C07312=1222.254,171.047,-53.911,-177.755,5.929,148.387
C07313=1222.250,171.296,-53.933,-177.752,5.931,148.387
C07314=1222.244,171.545,-53.955,-177.749,5.933,148.387
C07315=1222.240,171.794,-53.978,-177.747,5.934,148.386
C07316=1222.236,172.043,-54.000,-177.744,5.935,148.386
C07317=1222.230,172.292,-54.022,-177.742,5.936,148.385
C07318=1222.226,172.541,-54.044,-177.739,5.938,148.385
C07319=1222.221,172.789,-54.067,-177.736,5.940,148.384
C07320=1222.216,173.039,-54.089,-177.734,5.941,148.384
C07321=1222.212,173.288,-54.111,-177.732,5.943,148.384
C07322=1222.208,173.536,-54.134,-177.729,5.944,148.383
C07323=1222.203,173.786,-54.156,-177.726,5.945,148.383
C07324=1222.198,174.034,-54.179,-177.724,5.947,148.382
C07325=1222.194,174.283,-54.201,-177.721,5.949,148.382
C07326=1222.189,174.533,-54.223,-177.719,5.950,148.382
C07327=1222.184,174.781,-54.246,-177.716,5.951,148.381
C07328=1222.180,175.030,-54.268,-177.713,5.953,148.381
C07329=1222.174,175.279,-54.290,-177.711,5.954,148.380
C07330=1222.170,175.528,-54.313,-177.708,5.956,148.380
C07331=1222.165,175.778,-54.336,-177.706,5.957,148.379
C07332=1222.161,176.026,-54.358,-177.703,5.958,148.379
C07333=1222.157,176.275,-54.380,-177.701,5.960,148.379
C07334=1222.152,176.524,-54.403,-177.698,5.961,148.378
C07335=1222.147,176.773,-54.425,-177.696,5.963,148.378
C07336=1222.142,177.022,-54.448,-177.693,5.965,148.377
C07337=1222.138,177.271,-54.470,-177.691,5.966,148.377
C07338=1222.133,177.519,-54.493,-177.688,5.967,148.377
C07339=1222.128,177.769,-54.516,-177.685,5.969,148.376
C07340=1222.124,178.017,-54.538,-177.683,5.970,148.376
C07341=1222.119,178.266,-54.561,-177.680,5.972,148.375
C07342=1222.115,178.515,-54.583,-177.677,5.973,148.375
C07343=1222.110,178.765,-54.606,-177.675,5.974,148.375
C07344=1222.105,179.013,-54.628,-177.673,5.976,148.374
C07345=1222.101,179.262,-54.652,-177.669,5.978,148.374
C07346=1222.096,179.511,-54.674,-177.667,5.979,148.373
C07347=1222.092,179.760,-54.697,-177.665,5.981,148.373
C07348=1222.087,180.009,-54.719,-177.662,5.982,148.372
C07349=1222.082,180.258,-54.742,-177.659,5.984,148.372
C07350=1222.078,180.507,-54.765,-177.657,5.985,148.372
C07351=1222.073,180.756,-54.788,-177.654,5.987,148.371
C07352=1222.068,181.005,-54.811,-177.652,5.989,148.371
C07353=1222.064,181.254,-54.833,-177.649,5.990,148.370
C07354=1222.059,181.503,-54.856,-177.647,5.991,148.370
C07355=1222.054,181.751,-54.878,-177.644,5.993,148.370
C07356=1222.050,182.000,-54.902,-177.642,5.994,148.369
C07357=1222.045,182.249,-54.924,-177.639,5.996,148.369
C07358=1222.041,182.498,-54.947,-177.636,5.998,148.368
C07359=1222.037,182.747,-54.970,-177.634,5.999,148.368
C07360=1222.031,182.996,-54.992,-177.631,6.000,148.367
C07361=1222.026,183.245,-55.016,-177.628,6.002,148.367
C07362=1222.022,183.494,-55.038,-177.626,6.004,148.367
C07363=1222.018,183.743,-55.062,-177.624,6.005,148.366
C07364=1222.012,183.992,-55.084,-177.621,6.007,148.366
C07365=1222.008,184.240,-55.107,-177.618,6.009,148.366
C07366=1222.003,184.489,-55.130,-177.616,6.009,148.365
C07367=1221.999,184.738,-55.153,-177.613,6.011,148.365
C07368=1221.995,184.987,-55.176,-177.610,6.013,148.364
C07369=1221.989,185.257,-55.201,-177.608,6.015,148.364
C07370=1221.985,185.526,-55.226,-177.605,6.016,148.363
C07371=1221.980,185.796,-55.251,-177.602,6.018,148.363
C07372=1221.974,186.066,-55.276,-177.599,6.020,148.363
C07373=1221.970,186.315,-55.299,-177.597,6.021,148.362
C07374=1221.965,186.563,-55.322,-177.594,6.022,148.362
C07375=1221.960,186.812,-55.345,-177.592,6.024,148.361
C07376=1221.956,187.061,-55.368,-177.589,6.026,148.361
C07377=1221.951,187.310,-55.390,-177.587,6.027,148.361
C07378=1221.947,187.559,-55.414,-177.584,6.029,148.360
C07379=1221.942,187.809,-55.437,-177.581,6.031,148.360
C07380=1221.938,188.057,-55.460,-177.579,6.031,148.359
C07381=1221.933,188.306,-55.483,-177.576,6.033,148.359
C07382=1221.928,188.555,-55.506,-177.574,6.035,148.359
C07383=1221.923,188.804,-55.529,-177.571,6.037,148.358
C07384=1221.919,189.052,-55.552,-177.569,6.038,148.358
C07385=1221.915,189.301,-55.576,-177.566,6.040,148.358
C07386=1221.910,189.550,-55.599,-177.564,6.042,148.357
C07387=1221.905,189.799,-55.622,-177.560,6.043,148.357
C07388=1221.900,190.048,-55.646,-177.558,6.044,148.356
C07389=1221.896,190.296,-55.668,-177.556,6.046,148.356
C07390=1221.891,190.546,-55.691,-177.553,6.048,148.356
C07391=1221.887,190.795,-55.715,-177.550,6.050,148.355
C07392=1221.882,191.044,-55.738,-177.548,6.051,148.355
C07393=1221.877,191.293,-55.761,-177.546,6.052,148.355
C07394=1221.872,191.542,-55.785,-177.543,6.054,148.354
C07395=1221.869,191.790,-55.808,-177.540,6.056,148.354
C07396=1221.864,192.039,-55.832,-177.538,6.057,148.353
C07397=1221.859,192.288,-55.855,-177.535,6.059,148.353
C07398=1221.855,192.537,-55.878,-177.533,6.060,148.353
C07399=1221.850,192.786,-55.902,-177.530,6.062,148.352
C07400=1221.845,193.034,-55.925,-177.527,6.064,148.352
C07401=1221.840,193.283,-55.948,-177.525,6.065,148.351
C07402=1221.836,193.532,-55.972,-177.522,6.067,148.351
C07403=1221.831,193.781,-55.996,-177.519,6.069,148.351
C07404=1221.827,194.029,-56.018,-177.517,6.070,148.350
C07405=1221.822,194.278,-56.042,-177.515,6.071,148.350
C07406=1221.818,194.527,-56.065,-177.512,6.073,148.350
C07407=1221.813,194.776,-56.089,-177.509,6.075,148.349
C07408=1221.808,195.025,-56.112,-177.507,6.077,148.349
C07409=1221.804,195.274,-56.136,-177.504,6.079,148.348
C07410=1221.799,195.523,-56.159,-177.502,6.080,148.348
C07411=1221.795,195.771,-56.183,-177.499,6.081,148.348
C07412=1221.790,196.020,-56.207,-177.496,6.083,148.347
C07413=1221.785,196.269,-56.230,-177.494,6.085,148.347
C07414=1221.781,196.519,-56.253,-177.492,6.086,148.346
C07415=1221.776,196.767,-56.277,-177.489,6.088,148.346
C07416=1221.771,197.016,-56.301,-177.486,6.090,148.346
C07417=1221.767,197.265,-56.324,-177.484,6.091,148.345
C07418=1221.762,197.513,-56.348,-177.481,6.093,148.345
C07419=1221.758,197.762,-56.372,-177.479,6.094,148.345
C07420=1221.753,198.011,-56.395,-177.476,6.096,148.344
C07421=1221.749,198.260,-56.419,-177.474,6.098,148.344
C07422=1221.744,198.509,-56.442,-177.470,6.100,148.343
C07423=1221.739,198.757,-56.466,-177.468,6.101,148.343
C07424=1221.735,199.006,-56.490,-177.466,6.102,148.343
C07425=1221.730,199.255,-56.513,-177.463,6.104,148.342
C07426=1221.726,199.504,-56.538,-177.460,6.106,148.342
C07427=1221.722,199.754,-56.561,-177.458,6.108,148.342
C07428=1221.717,200.002,-56.585,-177.455,6.110,148.341
C07429=1221.712,200.251,-56.608,-177.453,6.112,148.341
C07430=1221.707,200.500,-56.633,-177.450,6.113,148.341
C07431=1221.703,200.749,-56.656,-177.448,6.114,148.340
C07432=1221.698,200.997,-56.680,-177.445,6.116,148.340
C07433=1221.694,201.246,-56.704,-177.443,6.118,148.340
C07434=1221.689,201.495,-56.728,-177.440,6.120,148.339
C07435=1221.684,201.744,-56.751,-177.437,6.121,148.339
C07436=1221.680,201.992,-56.775,-177.435,6.123,148.338
C07437=1221.675,202.241,-56.799,-177.432,6.124,148.338
C07438=1221.671,202.490,-56.824,-177.429,6.126,148.338
C07439=1221.666,202.740,-56.847,-177.427,6.128,148.337
C07440=1221.662,202.988,-56.871,-177.424,6.130,148.337
C07441=1221.657,203.237,-56.895,-177.422,6.131,148.337
C07442=1221.653,203.485,-56.919,-177.419,6.133,148.336
C07443=1221.648,203.734,-56.943,-177.417,6.135,148.336
C07444=1221.643,203.983,-56.967,-177.414,6.136,148.336
C07445=1221.639,204.232,-56.991,-177.411,6.138,148.335
C07446=1221.635,204.481,-57.015,-177.409,6.140,148.335
C07447=1221.630,204.730,-57.039,-177.407,6.141,148.335
C07448=1221.626,204.978,-57.063,-177.404,6.143,148.334
C07449=1221.620,205.227,-57.087,-177.401,6.145,148.334
C07450=1221.616,205.476,-57.111,-177.399,6.147,148.334
C07451=1221.611,205.724,-57.135,-177.396,6.149,148.333
C07452=1221.608,205.973,-57.159,-177.394,6.150,148.333
C07453=1221.602,206.223,-57.183,-177.391,6.152,148.333
C07454=1221.598,206.471,-57.207,-177.388,6.153,148.332
C07455=1221.593,206.720,-57.231,-177.386,6.155,148.332
C07456=1221.589,206.969,-57.255,-177.383,6.157,148.331
C07457=1221.584,207.218,-57.280,-177.380,6.158,148.331
C07458=1221.580,207.466,-57.304,-177.378,6.160,148.331
C07459=1221.575,207.715,-57.328,-177.375,6.162,148.330
C07460=1221.570,207.964,-57.352,-177.373,6.164,148.330
C07461=1221.565,208.213,-57.376,-177.370,6.165,148.330
C07462=1221.562,208.462,-57.400,-177.368,6.167,148.329
C07463=1221.557,208.710,-57.425,-177.365,6.169,148.329
C07464=1221.552,208.959,-57.449,-177.363,6.171,148.329
C07465=1221.548,209.207,-57.473,-177.360,6.172,148.328
C07466=1221.542,209.457,-57.497,-177.357,6.174,148.328
C07467=1221.538,209.706,-57.521,-177.355,6.176,148.328
C07468=1221.534,209.954,-57.546,-177.352,6.178,148.327
C07469=1221.529,210.203,-57.570,-177.349,6.180,148.327
C07470=1221.525,210.451,-57.594,-177.347,6.181,148.326
C07471=1221.520,210.701,-57.619,-177.345,6.183,148.326
C07472=1221.516,210.949,-57.643,-177.342,6.185,148.326
C07473=1221.510,211.219,-57.670,-177.339,6.186,148.325
C07474=1221.505,211.490,-57.696,-177.337,6.188,148.325
C07475=1221.501,211.761,-57.723,-177.334,6.191,148.325
C07476=1221.496,212.031,-57.749,-177.330,6.192,148.324
C07477=1221.491,212.280,-57.774,-177.328,6.194,148.324
C07478=1221.487,212.528,-57.798,-177.325,6.196,148.324
C07479=1221.482,212.777,-57.823,-177.323,6.197,148.323
C07480=1221.478,213.026,-57.847,-177.320,6.199,148.323
C07481=1221.473,213.274,-57.871,-177.318,6.201,148.323
C07482=1221.469,213.524,-57.896,-177.315,6.203,148.322
C07483=1221.464,213.772,-57.920,-177.313,6.205,148.322
C07484=1221.459,214.021,-57.945,-177.310,6.206,148.322
C07485=1221.455,214.270,-57.969,-177.307,6.208,148.321
C07486=1221.450,214.519,-57.994,-177.305,6.210,148.321
C07487=1221.446,214.767,-58.018,-177.302,6.212,148.321
C07488=1221.441,215.016,-58.043,-177.299,6.214,148.320
C07489=1221.437,215.265,-58.067,-177.297,6.216,148.320
C07490=1221.432,215.514,-58.092,-177.295,6.217,148.320
C07491=1221.428,215.762,-58.117,-177.293,6.219,148.319
C07492=1221.423,216.011,-58.142,-177.290,6.221,148.319
C07493=1221.418,216.259,-58.166,-177.287,6.223,148.319
C07494=1221.414,216.509,-58.191,-177.285,6.225,148.318
C07495=1221.409,216.757,-58.216,-177.282,6.226,148.318
C07496=1221.405,217.006,-58.240,-177.279,6.228,148.318
C07497=1221.400,217.255,-58.265,-177.277,6.230,148.317
C07498=1221.396,217.503,-58.289,-177.274,6.232,148.317
C07499=1221.391,217.752,-58.314,-177.271,6.234,148.317
C07500=1221.386,218.001,-58.339,-177.269,6.236,148.316
C07501=1221.382,218.250,-58.363,-177.266,6.237,148.316
C07502=1221.378,218.498,-58.389,-177.264,6.239,148.316
C07503=1221.373,218.747,-58.413,-177.262,6.240,148.315
C07504=1221.368,218.995,-58.438,-177.259,6.242,148.315
C07505=1221.364,219.245,-58.463,-177.256,6.244,148.315
C07506=1221.360,219.493,-58.488,-177.254,6.246,148.314
C07507=1221.355,219.742,-58.513,-177.251,6.248,148.314
C07508=1221.350,219.991,-58.537,-177.248,6.250,148.314
C07509=1221.347,220.239,-58.562,-177.246,6.252,148.313
C07510=1221.341,220.488,-58.587,-177.243,6.253,148.313
C07511=1221.336,220.737,-58.612,-177.240,6.255,148.313
C07512=1221.333,220.985,-58.637,-177.238,6.257,148.313
C07513=1221.328,221.234,-58.662,-177.236,6.259,148.312
C07514=1221.323,221.483,-58.687,-177.233,6.261,148.312
C07515=1221.319,221.731,-58.711,-177.230,6.263,148.312
C07516=1221.314,221.981,-58.736,-177.228,6.265,148.311
C07517=1221.310,222.229,-58.762,-177.225,6.267,148.311
C07518=1221.305,222.478,-58.787,-177.223,6.269,148.311
C07519=1221.301,222.727,-58.811,-177.220,6.270,148.310
C07520=1221.297,222.975,-58.837,-177.218,6.271,148.310
C07521=1221.291,223.224,-58.861,-177.215,6.273,148.310
C07522=1221.287,223.473,-58.887,-177.213,6.275,148.309
C07523=1221.283,223.721,-58.911,-177.210,6.277,148.309
C07524=1221.279,223.970,-58.937,-177.207,6.279,148.309
C07525=1221.273,224.219,-58.962,-177.205,6.281,148.309
C07526=1221.269,224.468,-58.987,-177.203,6.283,148.308
C07527=1221.265,224.716,-59.011,-177.200,6.285,148.308
C07528=1221.261,224.965,-59.037,-177.197,6.287,148.308
C07529=1221.255,225.214,-59.062,-177.195,6.288,148.307
C07530=1221.251,225.462,-59.088,-177.192,6.290,148.307
C07531=1221.246,225.711,-59.112,-177.189,6.292,148.307
C07532=1221.242,225.960,-59.138,-177.187,6.294,148.306
C07533=1221.238,226.208,-59.163,-177.184,6.296,148.306
C07534=1221.233,226.457,-59.188,-177.182,6.298,148.306
C07535=1221.228,226.705,-59.213,-177.179,6.300,148.306
C07536=1221.224,226.955,-59.238,-177.177,6.302,148.305
C07537=1221.219,227.203,-59.264,-177.174,6.304,148.305
C07538=1221.215,227.452,-59.289,-177.172,6.306,148.305
C07539=1221.210,227.701,-59.314,-177.169,6.307,148.304
C07540=1221.206,227.949,-59.339,-177.166,6.309,148.304
C07541=1221.202,228.198,-59.365,-177.164,6.311,148.304
C07542=1221.197,228.446,-59.390,-177.161,6.313,148.303
C07543=1221.193,228.695,-59.415,-177.159,6.315,148.303
C07544=1221.188,228.943,-59.441,-177.156,6.317,148.303
C07545=1221.183,229.193,-59.466,-177.154,6.319,148.303
C07546=1221.179,229.441,-59.492,-177.151,6.321,148.302
C07547=1221.174,229.690,-59.517,-177.149,6.322,148.302
C07548=1221.170,229.938,-59.543,-177.146,6.324,148.302
C07549=1221.165,230.187,-59.567,-177.144,6.326,148.301
C07550=1221.161,230.436,-59.593,-177.141,6.327,148.301
C07551=1221.156,230.685,-59.619,-177.139,6.330,148.301
C07552=1221.152,230.933,-59.644,-177.136,6.331,148.301
C07553=1221.147,231.182,-59.669,-177.134,6.333,148.300
C07554=1221.142,231.430,-59.695,-177.131,6.335,148.300
C07555=1221.138,231.679,-59.720,-177.128,6.337,148.300
C07556=1221.134,231.928,-59.746,-177.126,6.339,148.299
C07557=1221.129,232.176,-59.772,-177.124,6.341,148.299
C07558=1221.125,232.425,-59.797,-177.121,6.343,148.299
C07559=1221.120,232.674,-59.822,-177.118,6.345,148.299
C07560=1221.115,232.922,-59.848,-177.116,6.347,148.298
C07561=1221.111,233.171,-59.873,-177.113,6.349,148.298
C07562=1221.107,233.420,-59.899,-177.111,6.350,148.298
C07563=1221.102,233.668,-59.925,-177.108,6.353,148.297
C07564=1221.098,233.917,-59.950,-177.106,6.354,148.297
C07565=1221.094,234.166,-59.976,-177.103,6.356,148.297
C07566=1221.089,234.414,-60.002,-177.101,6.358,148.297
C07567=1221.085,234.663,-60.027,-177.098,6.360,148.296
C07568=1221.080,234.911,-60.053,-177.095,6.362,148.296
C07569=1221.076,235.159,-60.078,-177.093,6.364,148.296
C07570=1221.071,235.409,-60.105,-177.090,6.366,148.295
C07571=1221.066,235.657,-60.130,-177.088,6.368,148.295
C07572=1221.062,235.906,-60.156,-177.085,6.370,148.295
C07573=1221.057,236.154,-60.182,-177.083,6.372,148.295
C07574=1221.053,236.403,-60.207,-177.080,6.374,148.294
C07575=1221.049,236.652,-60.233,-177.078,6.376,148.294
C07576=1221.044,236.900,-60.259,-177.075,6.377,148.294
C07577=1221.039,237.172,-60.287,-177.072,6.380,148.293
C07578=1221.035,237.443,-60.315,-177.069,6.382,148.293
C07579=1221.029,237.715,-60.344,-177.067,6.384,148.293
C07580=1221.024,237.987,-60.372,-177.064,6.387,148.293
C07581=1221.020,238.235,-60.397,-177.061,6.388,148.292
C07582=1221.015,238.484,-60.423,-177.058,6.390,148.292
C07583=1221.011,238.732,-60.449,-177.056,6.393,148.292
C07584=1221.007,238.981,-60.475,-177.054,6.394,148.292
C07585=1221.002,239.230,-60.501,-177.051,6.396,148.291
C07586=1220.997,239.478,-60.527,-177.048,6.398,148.291
C07587=1220.993,239.727,-60.552,-177.046,6.400,148.291
C07588=1220.989,239.975,-60.578,-177.044,6.402,148.290
C07589=1220.984,240.224,-60.605,-177.041,6.404,148.290
C07590=1220.979,240.472,-60.631,-177.038,6.406,148.290
C07591=1220.975,240.721,-60.656,-177.036,6.408,148.290
C07592=1220.971,240.970,-60.682,-177.034,6.410,148.289
C07593=1220.966,241.218,-60.709,-177.031,6.412,148.289
C07594=1220.962,241.467,-60.735,-177.028,6.414,148.289
C07595=1220.957,241.715,-60.760,-177.026,6.416,148.289
C07596=1220.952,241.964,-60.787,-177.024,6.418,148.288
C07597=1220.948,242.212,-60.813,-177.021,6.420,148.288
C07598=1220.944,242.461,-60.839,-177.018,6.422,148.288
C07599=1220.939,242.710,-60.865,-177.016,6.423,148.287
C07600=1220.935,242.958,-60.892,-177.014,6.426,148.287
C07601=1220.930,243.206,-60.917,-177.011,6.427,148.287
C07602=1220.925,243.456,-60.943,-177.008,6.429,148.287
C07603=1220.921,243.704,-60.970,-177.005,6.432,148.286
C07604=1220.917,243.953,-60.996,-177.003,6.434,148.286
C07605=1220.912,244.202,-61.022,-177.001,6.436,148.286
C07606=1220.908,244.450,-61.048,-176.998,6.438,148.286
C07607=1220.904,244.699,-61.074,-176.995,6.440,148.285
C07608=1220.899,244.946,-61.101,-176.993,6.442,148.285
C07609=1220.895,245.195,-61.127,-176.991,6.444,148.285
C07610=1220.890,245.444,-61.153,-176.988,6.446,148.285
C07611=1220.886,245.693,-61.179,-176.985,6.448,148.284
C07612=1220.882,245.941,-61.205,-176.983,6.450,148.284
C07613=1220.877,246.190,-61.232,-176.981,6.452,148.284
C07614=1220.873,246.439,-61.258,-176.978,6.454,148.284
C07615=1220.868,246.687,-61.285,-176.975,6.455,148.283
C07616=1220.864,246.936,-61.311,-176.973,6.458,148.283
C07617=1220.859,247.184,-61.338,-176.971,6.459,148.283
C07618=1220.854,247.433,-61.363,-176.967,6.462,148.283
C07619=1220.850,247.681,-61.390,-176.965,6.464,148.283
C07620=1220.845,247.930,-61.416,-176.963,6.466,148.282
C07621=1220.841,248.178,-61.443,-176.960,6.468,148.282
C07622=1220.837,248.427,-61.470,-176.957,6.470,148.282
C07623=1220.832,248.676,-61.496,-176.955,6.472,148.282
C07624=1220.828,248.924,-61.522,-176.953,6.474,148.281
C07625=1220.823,249.173,-61.549,-176.950,6.476,148.281
C07626=1220.819,249.421,-61.575,-176.948,6.478,148.281
C07627=1220.814,249.670,-61.602,-176.945,6.480,148.281
C07628=1220.810,249.918,-61.628,-176.943,6.482,148.280
C07629=1220.806,250.167,-61.655,-176.941,6.484,148.280
C07630=1220.801,250.416,-61.681,-176.937,6.487,148.280
C07631=1220.797,250.664,-61.708,-176.935,6.489,148.280
C07632=1220.793,250.912,-61.734,-176.932,6.491,148.279
C07633=1220.788,251.162,-61.761,-176.930,6.493,148.279
C07634=1220.783,251.410,-61.788,-176.927,6.495,148.279
C07635=1220.779,251.658,-61.814,-176.925,6.496,148.279
C07636=1220.775,251.907,-61.841,-176.923,6.499,148.279
C07637=1220.770,252.156,-61.867,-176.920,6.501,148.278
C07638=1220.766,252.404,-61.894,-176.917,6.502,148.278
C07639=1220.761,252.653,-61.921,-176.915,6.505,148.278
C07640=1220.757,252.901,-61.948,-176.912,6.507,148.278
C07641=1220.752,253.150,-61.974,-176.909,6.509,148.277
C07642=1220.748,253.398,-62.001,-176.907,6.511,148.277
C07643=1220.744,253.647,-62.028,-176.905,6.513,148.277
C07644=1220.739,253.895,-62.055,-176.902,6.515,148.277
C07645=1220.735,254.143,-62.081,-176.900,6.517,148.276
C07646=1220.730,254.392,-62.107,-176.897,6.519,148.276
C07647=1220.725,254.641,-62.135,-176.895,6.521,148.276
C07648=1220.721,254.889,-62.161,-176.892,6.524,148.276
C07649=1220.717,255.137,-62.188,-176.889,6.526,148.276
C07650=1220.712,255.386,-62.215,-176.887,6.528,148.275
C07651=1220.707,255.634,-62.242,-176.885,6.530,148.275
C07652=1220.704,255.883,-62.269,-176.882,6.532,148.275
C07653=1220.699,256.131,-62.296,-176.880,6.534,148.275
C07654=1220.694,256.380,-62.323,-176.877,6.536,148.274
C07655=1220.691,256.629,-62.350,-176.874,6.539,148.274
C07656=1220.686,256.878,-62.376,-176.872,6.541,148.274
C07657=1220.681,257.126,-62.403,-176.869,6.543,148.274
C07658=1220.677,257.375,-62.430,-176.867,6.545,148.273
C07659=1220.673,257.623,-62.457,-176.865,6.547,148.273
C07660=1220.668,257.871,-62.484,-176.862,6.549,148.273
C07661=1220.663,258.120,-62.511,-176.860,6.551,148.273
C07662=1220.659,258.368,-62.538,-176.857,6.553,148.273
C07663=1220.654,258.617,-62.565,-176.854,6.556,148.272
C07664=1220.651,258.866,-62.592,-176.852,6.558,148.272
C07665=1220.646,259.114,-62.619,-176.849,6.560,148.272
C07666=1220.642,259.362,-62.646,-176.847,6.561,148.272
C07667=1220.637,259.611,-62.674,-176.845,6.564,148.272
C07668=1220.632,259.859,-62.701,-176.842,6.566,148.271
C07669=1220.628,260.108,-62.728,-176.839,6.569,148.271
C07670=1220.624,260.356,-62.754,-176.837,6.570,148.271
C07671=1220.620,260.605,-62.782,-176.834,6.572,148.271
C07672=1220.615,260.853,-62.809,-176.832,6.575,148.271
C07673=1220.611,261.102,-62.836,-176.829,6.576,148.270
C07674=1220.606,261.350,-62.863,-176.827,6.579,148.270
C07675=1220.602,261.598,-62.890,-176.824,6.581,148.270
C07676=1220.597,261.847,-62.918,-176.822,6.583,148.270
C07677=1220.593,262.096,-62.945,-176.819,6.585,148.270
C07678=1220.589,262.344,-62.971,-176.817,6.587,148.269
C07679=1220.584,262.593,-62.999,-176.815,6.589,148.269
C07680=1220.580,262.841,-63.026,-176.812,6.591,148.269
C07681=1220.574,263.114,-63.056,-176.809,6.594,148.269
C07682=1220.570,263.386,-63.086,-176.807,6.596,148.269
C07683=1220.565,263.659,-63.116,-176.804,6.599,148.268
C07684=1220.561,263.932,-63.146,-176.801,6.601,148.268
C07685=1220.556,264.180,-63.173,-176.798,6.604,148.268
C07686=1220.552,264.428,-63.201,-176.796,6.606,148.268
C07687=1220.547,264.677,-63.228,-176.793,6.608,148.267
C07688=1220.543,264.926,-63.255,-176.791,6.610,148.267
C07689=1220.539,265.174,-63.283,-176.788,6.612,148.267
C07690=1220.534,265.422,-63.310,-176.786,6.614,148.267
C07691=1220.529,265.671,-63.337,-176.783,6.617,148.267
C07692=1220.525,265.919,-63.365,-176.781,6.619,148.267
C07693=1220.521,266.168,-63.392,-176.778,6.621,148.266
C07694=1220.516,266.416,-63.419,-176.776,6.623,148.266
C07695=1220.512,266.664,-63.447,-176.774,6.625,148.266
C07696=1220.508,266.913,-63.475,-176.771,6.628,148.266
C07697=1220.503,267.161,-63.502,-176.768,6.630,148.266
C07698=1220.499,267.410,-63.530,-176.766,6.632,148.265
C07699=1220.493,267.658,-63.557,-176.764,6.634,148.265
C07700=1220.490,267.907,-63.585,-176.761,6.636,148.265
C07701=1220.485,268.156,-63.612,-176.758,6.639,148.265
C07702=1220.481,268.403,-63.640,-176.756,6.641,148.265
C07703=1220.477,268.653,-63.668,-176.754,6.643,148.265
C07704=1220.472,268.901,-63.695,-176.751,6.645,148.264
C07705=1220.468,269.149,-63.722,-176.748,6.648,148.264
C07706=1220.464,269.398,-63.751,-176.746,6.650,148.264
C07707=1220.459,269.646,-63.778,-176.744,6.652,148.264
C07708=1220.454,269.894,-63.806,-176.741,6.654,148.264
C07709=1220.450,270.143,-63.834,-176.739,6.656,148.263
C07710=1220.446,270.391,-63.861,-176.736,6.659,148.263
C07711=1220.441,270.639,-63.889,-176.734,6.661,148.263
C07712=1220.437,270.888,-63.916,-176.731,6.663,148.263
C07713=1220.433,271.136,-63.944,-176.729,6.665,148.263
C07714=1220.428,271.385,-63.971,-176.726,6.668,148.262
C07715=1220.424,271.634,-64.000,-176.724,6.670,148.262
C07716=1220.419,271.882,-64.028,-176.721,6.672,148.262
C07717=1220.415,272.130,-64.055,-176.719,6.674,148.262
C07718=1220.411,272.379,-64.083,-176.716,6.676,148.262
C07719=1220.406,272.627,-64.111,-176.714,6.679,148.262
C07720=1220.401,272.875,-64.138,-176.711,6.681,148.261
C07721=1220.397,273.124,-64.167,-176.709,6.683,148.261
C07722=1220.393,273.372,-64.194,-176.706,6.685,148.261
C07723=1220.389,273.620,-64.222,-176.704,6.688,148.261
C07724=1220.384,273.869,-64.250,-176.701,6.690,148.261
C07725=1220.380,274.117,-64.278,-176.699,6.692,148.261
C07726=1220.376,274.366,-64.306,-176.697,6.694,148.261
C07727=1220.371,274.614,-64.334,-176.694,6.697,148.260
C07728=1220.367,274.863,-64.362,-176.691,6.699,148.260
C07729=1220.362,275.111,-64.390,-176.689,6.701,148.260
C07730=1220.359,275.359,-64.418,-176.687,6.703,148.260
C07731=1220.354,275.608,-64.446,-176.684,6.706,148.260
C07732=1220.349,275.855,-64.474,-176.681,6.708,148.260
C07733=1220.345,276.105,-64.501,-176.679,6.710,148.259
C07734=1220.340,276.353,-64.530,-176.677,6.712,148.259
C07735=1220.336,276.601,-64.558,-176.674,6.715,148.259
C07736=1220.332,276.849,-64.586,-176.671,6.717,148.259
C07737=1220.327,277.098,-64.614,-176.669,6.719,148.259
C07738=1220.323,277.346,-64.642,-176.666,6.722,148.259
C07739=1220.319,277.595,-64.670,-176.664,6.724,148.258
C07740=1220.314,277.843,-64.699,-176.661,6.726,148.258
C07741=1220.310,278.092,-64.726,-176.659,6.728,148.258
C07742=1220.305,278.340,-64.754,-176.657,6.731,148.258
C07743=1220.301,278.589,-64.783,-176.654,6.733,148.258
C07744=1220.297,278.837,-64.810,-176.652,6.735,148.258
C07745=1220.293,279.086,-64.839,-176.649,6.737,148.257
C07746=1220.288,279.333,-64.867,-176.647,6.740,148.257
C07747=1220.284,279.582,-64.896,-176.644,6.743,148.257
C07748=1220.279,279.830,-64.923,-176.642,6.744,148.257
C07749=1220.275,280.079,-64.952,-176.639,6.748,148.257
C07750=1220.270,280.327,-64.980,-176.637,6.749,148.257
C07751=1220.267,280.576,-65.008,-176.634,6.752,148.257
C07752=1220.262,280.824,-65.036,-176.632,6.754,148.257
C07753=1220.258,281.072,-65.065,-176.629,6.757,148.256
C07754=1220.253,281.320,-65.094,-176.627,6.759,148.256
C07755=1220.249,281.568,-65.122,-176.625,6.761,148.256
C07756=1220.244,281.817,-65.150,-176.622,6.764,148.256
C07757=1220.241,282.065,-65.178,-176.620,6.766,148.256
C07758=1220.235,282.313,-65.207,-176.617,6.768,148.256
C07759=1220.232,282.562,-65.235,-176.615,6.770,148.256
C07760=1220.227,282.811,-65.264,-176.612,6.773,148.256
C07761=1220.223,283.059,-65.291,-176.610,6.775,148.255
C07762=1220.219,283.307,-65.321,-176.608,6.777,148.255
C07763=1220.214,283.555,-65.349,-176.605,6.780,148.255
C07764=1220.210,283.804,-65.377,-176.602,6.782,148.255
C07765=1220.205,284.052,-65.406,-176.600,6.784,148.255
C07766=1220.201,284.301,-65.434,-176.598,6.787,148.255
C07767=1220.197,284.549,-65.463,-176.595,6.789,148.254
C07768=1220.192,284.797,-65.491,-176.593,6.791,148.254
C07769=1220.188,285.046,-65.520,-176.591,6.794,148.254
C07770=1220.183,285.294,-65.548,-176.588,6.796,148.254
C07771=1220.179,285.542,-65.577,-176.585,6.799,148.254
C07772=1220.175,285.791,-65.606,-176.583,6.801,148.254
C07773=1220.170,286.039,-65.634,-176.580,6.803,148.254
C07774=1220.166,286.287,-65.663,-176.578,6.806,148.254
C07775=1220.162,286.536,-65.692,-176.576,6.808,148.254
C07776=1220.158,286.783,-65.720,-176.573,6.811,148.253
C07777=1220.153,287.032,-65.749,-176.571,6.813,148.253
C07778=1220.148,287.280,-65.777,-176.569,6.815,148.253
C07779=1220.145,287.529,-65.805,-176.566,6.818,148.253
C07780=1220.140,287.777,-65.835,-176.563,6.820,148.253
C07781=1220.135,288.025,-65.863,-176.561,6.822,148.253
C07782=1220.131,288.274,-65.892,-176.558,6.825,148.253
C07783=1220.127,288.522,-65.921,-176.556,6.827,148.253
C07784=1220.122,288.770,-65.949,-176.554,6.829,148.253
C07785=1220.117,289.044,-65.981,-176.551,6.832,148.252
C07786=1220.113,289.318,-66.013,-176.548,6.835,148.252
C07787=1220.108,289.592,-66.045,-176.546,6.837,148.252
C07788=1220.103,289.867,-66.077,-176.543,6.840,148.252
C07789=1220.099,290.115,-66.106,-176.541,6.842,148.252
C07790=1220.094,290.363,-66.134,-176.538,6.845,148.252
C07791=1220.091,290.611,-66.163,-176.536,6.847,148.252
C07792=1220.086,290.860,-66.192,-176.533,6.849,148.252
C07793=1220.082,291.108,-66.221,-176.530,6.852,148.252
C07794=1220.077,291.357,-66.250,-176.528,6.855,148.251
C07795=1220.073,291.605,-66.279,-176.526,6.857,148.251
C07796=1220.069,291.853,-66.307,-176.524,6.860,148.251
C07797=1220.064,292.101,-66.336,-176.521,6.862,148.251
C07798=1220.060,292.349,-66.366,-176.519,6.864,148.251
C07799=1220.056,292.598,-66.395,-176.516,6.867,148.251
C07800=1220.051,292.846,-66.424,-176.514,6.869,148.251
C07801=1220.047,293.094,-66.452,-176.511,6.872,148.251
C07802=1220.043,293.343,-66.481,-176.509,6.874,148.251
C07803=1220.039,293.591,-66.511,-176.507,6.876,148.251
C07804=1220.034,293.840,-66.540,-176.504,6.879,148.251
C07805=1220.030,294.088,-66.569,-176.502,6.882,148.251
C07806=1220.025,294.336,-66.598,-176.499,6.883,148.250
C07807=1220.021,294.584,-66.628,-176.497,6.887,148.250
C07808=1220.017,294.832,-66.656,-176.495,6.889,148.250
C07809=1220.013,295.081,-66.685,-176.492,6.891,148.250
C07810=1220.008,295.328,-66.714,-176.490,6.894,148.250
C07811=1220.004,295.577,-66.743,-176.487,6.896,148.250
C07812=1220.000,295.825,-66.772,-176.485,6.898,148.250
C07813=1219.995,296.074,-66.802,-176.482,6.901,148.250
C07814=1219.991,296.322,-66.831,-176.480,6.903,148.250
C07815=1219.987,296.570,-66.861,-176.478,6.906,148.250
C07816=1219.982,296.818,-66.889,-176.475,6.909,148.250
C07817=1219.978,297.067,-66.919,-176.473,6.910,148.249
C07818=1219.974,297.315,-66.948,-176.470,6.914,148.249
C07819=1219.969,297.563,-66.978,-176.468,6.916,148.249
C07820=1219.965,297.811,-67.007,-176.466,6.918,148.249
C07821=1219.961,298.060,-67.036,-176.463,6.921,148.249
C07822=1219.956,298.308,-67.065,-176.461,6.923,148.249
C07823=1219.952,298.556,-67.094,-176.459,6.926,148.249
C07824=1219.948,298.804,-67.124,-176.456,6.928,148.249
C07825=1219.943,299.053,-67.153,-176.454,6.930,148.249
C07826=1219.939,299.301,-67.183,-176.451,6.933,148.249
C07827=1219.935,299.549,-67.212,-176.449,6.936,148.249
C07828=1219.931,299.797,-67.242,-176.447,6.938,148.249
C07829=1219.926,300.045,-67.271,-176.444,6.941,148.249
C07830=1219.922,300.293,-67.300,-176.442,6.943,148.249
C07831=1219.918,300.542,-67.330,-176.439,6.946,148.249
C07832=1219.914,300.790,-67.359,-176.437,6.948,148.248
C07833=1219.909,301.038,-67.388,-176.435,6.950,148.248
C07834=1219.905,301.286,-67.418,-176.432,6.953,148.248
C07835=1219.901,301.535,-67.447,-176.430,6.955,148.248
C07836=1219.896,301.783,-67.477,-176.427,6.959,148.248
C07837=1219.892,302.032,-67.507,-176.425,6.961,148.248
C07838=1219.888,302.280,-67.536,-176.423,6.963,148.248
C07839=1219.884,302.528,-67.566,-176.420,6.966,148.248
C07840=1219.879,302.776,-67.595,-176.418,6.968,148.248
C07841=1219.875,303.024,-67.624,-176.416,6.971,148.248
C07842=1219.870,303.272,-67.654,-176.414,6.973,148.248
C07843=1219.865,303.521,-67.684,-176.411,6.976,148.248
C07844=1219.862,303.768,-67.714,-176.409,6.979,148.248
C07845=1219.857,304.017,-67.743,-176.407,6.981,148.248
C07846=1219.853,304.265,-67.773,-176.404,6.984,148.248
C07847=1219.849,304.513,-67.802,-176.402,6.986,148.248
C07848=1219.844,304.762,-67.832,-176.399,6.988,148.247
C07849=1219.840,305.010,-67.862,-176.397,6.991,148.247
C07850=1219.836,305.258,-67.892,-176.394,6.993,148.247
C07851=1219.832,305.506,-67.921,-176.392,6.996,148.247
C07852=1219.828,305.754,-67.951,-176.390,6.999,148.247
C07853=1219.823,306.003,-67.981,-176.388,7.001,148.247
C07854=1219.819,306.250,-68.011,-176.385,7.004,148.247
C07855=1219.815,306.499,-68.041,-176.383,7.006,148.247
C07856=1219.811,306.747,-68.070,-176.380,7.009,148.247
C07857=1219.806,306.996,-68.100,-176.378,7.011,148.247
C07858=1219.802,307.243,-68.130,-176.376,7.014,148.247
C07859=1219.798,307.491,-68.160,-176.373,7.017,148.247
C07860=1219.793,307.740,-68.190,-176.371,7.019,148.247
C07861=1219.789,307.988,-68.220,-176.368,7.022,148.247
C07862=1219.785,308.236,-68.249,-176.367,7.024,148.247
C07863=1219.780,308.485,-68.279,-176.365,7.027,148.247
C07864=1219.776,308.732,-68.310,-176.362,7.030,148.247
C07865=1219.772,308.980,-68.339,-176.360,7.032,148.247
C07866=1219.767,309.229,-68.369,-176.357,7.035,148.247
C07867=1219.763,309.477,-68.399,-176.355,7.037,148.247
C07868=1219.759,309.725,-68.429,-176.352,7.040,148.247
C07869=1219.754,309.973,-68.459,-176.350,7.042,148.247
C07870=1219.750,310.221,-68.489,-176.348,7.045,148.247
C07871=1219.746,310.469,-68.519,-176.346,7.048,148.247
C07872=1219.741,310.717,-68.549,-176.343,7.050,148.247
C07873=1219.737,310.966,-68.579,-176.341,7.053,148.247
C07874=1219.733,311.214,-68.610,-176.339,7.055,148.247
C07875=1219.729,311.463,-68.639,-176.336,7.058,148.247
C07876=1219.725,311.710,-68.669,-176.334,7.060,148.247
C07877=1219.720,311.959,-68.699,-176.332,7.063,148.247
C07878=1219.716,312.206,-68.730,-176.330,7.066,148.247
C07879=1219.711,312.454,-68.760,-176.328,7.068,148.247
C07880=1219.707,312.703,-68.790,-176.325,7.071,148.247
C07881=1219.703,312.951,-68.821,-176.323,7.073,148.247
C07882=1219.698,313.199,-68.850,-176.321,7.076,148.247
C07883=1219.695,313.447,-68.881,-176.318,7.079,148.247
C07884=1219.690,313.696,-68.911,-176.316,7.081,148.247
C07885=1219.686,313.943,-68.941,-176.314,7.084,148.247
C07886=1219.682,314.191,-68.971,-176.312,7.086,148.247
C07887=1219.678,314.440,-69.001,-176.309,7.090,148.247
C07888=1219.673,314.688,-69.032,-176.307,7.092,148.247
C07889=1219.668,314.964,-69.065,-176.304,7.095,148.247
C07890=1219.664,315.240,-69.099,-176.301,7.098,148.247
C07891=1219.659,315.516,-69.133,-176.299,7.100,148.247
C07892=1219.654,315.792,-69.167,-176.297,7.103,148.247
C07893=1219.650,316.039,-69.197,-176.294,7.106,148.247
C07894=1219.645,316.288,-69.227,-176.292,7.109,148.247
C07895=1219.641,316.536,-69.257,-176.290,7.112,148.247
C07896=1219.637,316.784,-69.288,-176.288,7.114,148.247
C07897=1219.633,317.032,-69.318,-176.285,7.116,148.247
C07898=1219.628,317.280,-69.349,-176.283,7.119,148.247
C07899=1219.625,317.528,-69.379,-176.281,7.122,148.247
C07900=1219.620,317.776,-69.409,-176.279,7.125,148.247
C07901=1219.616,318.025,-69.441,-176.276,7.127,148.247
C07902=1219.612,318.272,-69.471,-176.274,7.130,148.247
C07903=1219.607,318.521,-69.501,-176.272,7.133,148.247
C07904=1219.603,318.769,-69.532,-176.269,7.136,148.247
C07905=1219.599,319.017,-69.562,-176.267,7.138,148.247
C07906=1219.595,319.265,-69.593,-176.265,7.140,148.247
C07907=1219.591,319.513,-69.623,-176.263,7.143,148.247
C07908=1219.586,319.761,-69.654,-176.261,7.146,148.247
C07909=1219.582,320.009,-69.685,-176.258,7.149,148.247
C07910=1219.578,320.257,-69.715,-176.256,7.151,148.247
C07911=1219.573,320.506,-69.745,-176.254,7.154,148.247
C07912=1219.569,320.754,-69.776,-176.252,7.156,148.247
C07913=1219.565,321.001,-69.806,-176.250,7.159,148.247
C07914=1219.561,321.250,-69.837,-176.247,7.162,148.247
C07915=1219.556,321.498,-69.868,-176.245,7.164,148.247
C07916=1219.552,321.746,-69.899,-176.243,7.167,148.247
C07917=1219.548,321.994,-69.929,-176.241,7.169,148.247
C07918=1219.544,322.242,-69.960,-176.238,7.173,148.248
C07919=1219.539,322.490,-69.991,-176.236,7.175,148.248
C07920=1219.535,322.738,-70.021,-176.234,7.178,148.248
C07921=1219.531,322.986,-70.052,-176.232,7.181,148.248
C07922=1219.527,323.234,-70.083,-176.230,7.183,148.248
C07923=1219.522,323.482,-70.114,-176.227,7.186,148.248
C07924=1219.519,323.730,-70.145,-176.226,7.188,148.248
C07925=1219.514,323.978,-70.176,-176.223,7.191,148.248
C07926=1219.510,324.226,-70.206,-176.221,7.194,148.248
C07927=1219.506,324.475,-70.238,-176.219,7.197,148.248
C07928=1219.501,324.723,-70.268,-176.217,7.199,148.248
C07929=1219.497,324.970,-70.298,-176.214,7.201,148.248
C07930=1219.493,325.219,-70.330,-176.212,7.205,148.248
C07931=1219.489,325.467,-70.360,-176.210,7.207,148.248
C07932=1219.484,325.715,-70.391,-176.208,7.210,148.248
C07933=1219.480,325.963,-70.423,-176.206,7.213,148.248
C07934=1219.476,326.211,-70.454,-176.203,7.216,148.248
C07935=1219.472,326.459,-70.484,-176.202,7.218,148.248
C07936=1219.468,326.707,-70.515,-176.199,7.221,148.248
C07937=1219.463,326.955,-70.546,-176.197,7.224,148.249
C07938=1219.459,327.202,-70.577,-176.195,7.226,148.249
C07939=1219.455,327.451,-70.608,-176.193,7.229,148.249
C07940=1219.450,327.699,-70.639,-176.191,7.232,148.249
C07941=1219.446,327.948,-70.670,-176.188,7.235,148.249
C07942=1219.442,328.195,-70.702,-176.187,7.237,148.249
C07943=1219.438,328.443,-70.732,-176.184,7.240,148.249
C07944=1219.434,328.691,-70.763,-176.182,7.243,148.249
C07945=1219.430,328.939,-70.795,-176.180,7.246,148.249
C07946=1219.426,329.187,-70.826,-176.178,7.248,148.249
C07947=1219.421,329.435,-70.856,-176.176,7.250,148.249
C07948=1219.417,329.683,-70.888,-176.174,7.254,148.249
C07949=1219.413,329.931,-70.919,-176.172,7.256,148.249
C07950=1219.408,330.179,-70.950,-176.169,7.259,148.250
C07951=1219.405,330.427,-70.982,-176.167,7.262,148.250
C07952=1219.400,330.675,-71.012,-176.165,7.265,148.250
C07953=1219.396,330.923,-71.044,-176.163,7.267,148.250
C07954=1219.392,331.171,-71.075,-176.161,7.270,148.250
C07955=1219.387,331.419,-71.106,-176.159,7.273,148.250
C07956=1219.383,331.667,-71.138,-176.157,7.275,148.250
C07957=1219.379,331.915,-71.168,-176.154,7.278,148.250
C07958=1219.375,332.163,-71.200,-176.153,7.281,148.250
C07959=1219.370,332.411,-71.231,-176.150,7.284,148.250
C07960=1219.367,332.659,-71.263,-176.148,7.286,148.251
C07961=1219.362,332.907,-71.294,-176.147,7.289,148.251
C07962=1219.358,333.155,-71.325,-176.144,7.292,148.251
C07963=1219.354,333.403,-71.356,-176.142,7.295,148.251
C07964=1219.350,333.651,-71.388,-176.140,7.298,148.251
C07965=1219.345,333.899,-71.419,-176.138,7.300,148.251
C07966=1219.341,334.148,-71.451,-176.136,7.303,148.251
C07967=1219.336,334.396,-71.482,-176.134,7.306,148.251
C07968=1219.333,334.644,-71.514,-176.132,7.309,148.251
C07969=1219.328,334.892,-71.545,-176.130,7.311,148.251
C07970=1219.324,335.140,-71.577,-176.128,7.314,148.252
C07971=1219.320,335.387,-71.608,-176.126,7.317,148.252
C07972=1219.316,335.636,-71.639,-176.124,7.319,148.252
C07973=1219.312,335.883,-71.671,-176.121,7.323,148.252
C07974=1219.308,336.131,-71.702,-176.119,7.325,148.252
C07975=1219.303,336.379,-71.734,-176.117,7.328,148.252
C07976=1219.299,336.627,-71.766,-176.116,7.331,148.252
C07977=1219.295,336.875,-71.797,-176.113,7.333,148.252
C07978=1219.291,337.123,-71.828,-176.111,7.336,148.253
C07979=1219.286,337.371,-71.860,-176.110,7.339,148.253
C07980=1219.283,337.619,-71.892,-176.107,7.342,148.253
C07981=1219.277,337.867,-71.923,-176.105,7.345,148.253
C07982=1219.274,338.115,-71.955,-176.104,7.347,148.253
C07983=1219.270,338.363,-71.987,-176.101,7.350,148.253
C07984=1219.266,338.610,-72.018,-176.099,7.353,148.253
C07985=1219.262,338.859,-72.049,-176.097,7.356,148.254
C07986=1219.257,339.107,-72.081,-176.096,7.358,148.254
C07987=1219.253,339.355,-72.113,-176.093,7.362,148.254
C07988=1219.249,339.603,-72.145,-176.091,7.364,148.254
C07989=1219.244,339.851,-72.176,-176.090,7.367,148.254
C07990=1219.240,340.099,-72.208,-176.087,7.370,148.254
C07991=1219.236,340.346,-72.240,-176.086,7.372,148.254
C07992=1219.232,340.594,-72.272,-176.083,7.376,148.254
C07993=1219.228,340.872,-72.307,-176.081,7.378,148.255
C07994=1219.222,341.150,-72.343,-176.079,7.381,148.255
C07995=1219.218,341.428,-72.378,-176.077,7.385,148.255
C07996=1219.213,341.706,-72.414,-176.074,7.388,148.255
C07997=1219.209,341.954,-72.446,-176.073,7.390,148.255
C07998=1219.205,342.202,-72.477,-176.071,7.394,148.256
C07999=1219.200,342.450,-72.509,-176.069,7.396,148.256
C08000=1219.196,342.697,-72.541,-176.067,7.400,148.256
C08001=1219.192,342.945,-72.573,-176.065,7.402,148.256
C08002=1219.188,343.194,-72.605,-176.063,7.404,148.256
C08003=1219.183,343.441,-72.637,-176.061,7.408,148.256
C08004=1219.180,343.689,-72.669,-176.059,7.410,148.257
C08005=1219.175,343.938,-72.701,-176.057,7.414,148.257
C08006=1219.171,344.185,-72.732,-176.055,7.416,148.257
C08007=1219.167,344.433,-72.765,-176.054,7.419,148.257
C08008=1219.163,344.681,-72.797,-176.052,7.422,148.257
C08009=1219.159,344.929,-72.828,-176.049,7.424,148.257
C08010=1219.154,345.177,-72.861,-176.047,7.428,148.258
C08011=1219.150,345.425,-72.893,-176.046,7.430,148.258
C08012=1219.145,345.673,-72.925,-176.044,7.433,148.258
C08013=1219.142,345.921,-72.956,-176.042,7.436,148.258
C08014=1219.138,346.168,-72.989,-176.040,7.438,148.258
C08015=1219.133,346.416,-73.021,-176.038,7.442,148.259
C08016=1219.129,346.664,-73.053,-176.036,7.444,148.259
C08017=1219.125,346.912,-73.085,-176.035,7.447,148.259
C08018=1219.121,347.160,-73.117,-176.032,7.450,148.259
C08019=1219.116,347.408,-73.149,-176.031,7.453,148.259
C08020=1219.113,347.656,-73.181,-176.029,7.455,148.259
C08021=1219.108,347.904,-73.214,-176.027,7.459,148.260
C08022=1219.104,348.151,-73.246,-176.025,7.461,148.260
C08023=1219.100,348.399,-73.278,-176.023,7.464,148.260
C08024=1219.096,348.647,-73.310,-176.022,7.467,148.260
C08025=1219.092,348.896,-73.343,-176.020,7.470,148.260
C08026=1219.087,349.143,-73.374,-176.018,7.473,148.261
C08027=1219.083,349.391,-73.407,-176.016,7.475,148.261
C08028=1219.079,349.639,-73.439,-176.014,7.478,148.261
C08029=1219.075,349.887,-73.471,-176.012,7.481,148.261
C08030=1219.071,350.134,-73.503,-176.011,7.484,148.261
C08031=1219.066,350.382,-73.536,-176.008,7.487,148.262
C08032=1219.063,350.630,-73.568,-176.007,7.490,148.262
C08033=1219.058,350.879,-73.600,-176.005,7.492,148.262
C08034=1219.054,351.126,-73.632,-176.003,7.496,148.262
C08035=1219.050,351.374,-73.665,-176.001,7.498,148.262
C08036=1219.045,351.622,-73.697,-176.000,7.501,148.263
C08037=1219.042,351.870,-73.729,-175.998,7.504,148.263
C08038=1219.038,352.118,-73.762,-175.996,7.507,148.263
C08039=1219.033,352.365,-73.794,-175.995,7.509,148.263
C08040=1219.029,352.613,-73.827,-175.992,7.513,148.264
C08041=1219.025,352.861,-73.860,-175.991,7.515,148.264
C08042=1219.021,353.109,-73.891,-175.989,7.518,148.264
C08043=1219.017,353.357,-73.925,-175.987,7.521,148.264
C08044=1219.013,353.604,-73.956,-175.986,7.524,148.265
C08045=1219.008,353.852,-73.989,-175.984,7.527,148.265
C08046=1219.004,354.100,-74.022,-175.982,7.530,148.265
C08047=1219.000,354.348,-74.053,-175.980,7.532,148.265
C08048=1218.996,354.596,-74.087,-175.978,7.536,148.266
C08049=1218.992,354.845,-74.119,-175.977,7.538,148.266
C08050=1218.988,355.091,-74.151,-175.975,7.541,148.266
C08051=1218.983,355.340,-74.184,-175.973,7.544,148.266
C08052=1218.979,355.587,-74.217,-175.971,7.547,148.266
C08053=1218.975,355.835,-74.249,-175.970,7.549,148.267
C08054=1218.971,356.083,-74.282,-175.968,7.553,148.267
C08055=1218.967,356.331,-74.314,-175.966,7.556,148.267
C08056=1218.962,356.578,-74.347,-175.965,7.558,148.267
C08057=1218.958,356.826,-74.379,-175.963,7.561,148.268
C08058=1218.954,357.074,-74.412,-175.961,7.564,148.268
C08059=1218.950,357.322,-74.445,-175.960,7.567,148.268
C08060=1218.946,357.570,-74.477,-175.958,7.569,148.268
C08061=1218.942,357.818,-74.510,-175.956,7.573,148.269
C08062=1218.938,358.066,-74.543,-175.955,7.575,148.269
C08063=1218.934,358.314,-74.576,-175.953,7.578,148.269
C08064=1218.930,358.562,-74.608,-175.951,7.582,148.270
C08065=1218.925,358.809,-74.640,-175.950,7.584,148.270
C08066=1218.921,359.057,-74.674,-175.948,7.587,148.270
C08067=1218.917,359.305,-74.706,-175.946,7.590,148.271
C08068=1218.913,359.553,-74.739,-175.945,7.593,148.271
C08069=1218.909,359.800,-74.772,-175.943,7.595,148.271
C08070=1218.905,360.048,-74.804,-175.942,7.598,148.271
C08071=1218.901,360.296,-74.837,-175.940,7.602,148.272
C08072=1218.896,360.544,-74.871,-175.939,7.604,148.272
C08073=1218.892,360.792,-74.904,-175.937,7.607,148.272
C08074=1218.889,361.040,-74.936,-175.935,7.610,148.272
C08075=1218.884,361.287,-74.969,-175.934,7.613,148.273
C08076=1218.880,361.535,-75.002,-175.932,7.616,148.273
C08077=1218.876,361.783,-75.034,-175.931,7.618,148.273
C08078=1218.872,362.031,-75.067,-175.929,7.622,148.274
C08079=1218.868,362.279,-75.101,-175.927,7.625,148.274
C08080=1218.864,362.526,-75.133,-175.926,7.627,148.274
C08081=1218.859,362.773,-75.166,-175.925,7.630,148.275
C08082=1218.855,363.022,-75.198,-175.922,7.633,148.275
C08083=1218.851,363.269,-75.232,-175.921,7.636,148.275
C08084=1218.847,363.517,-75.265,-175.920,7.639,148.275
C08085=1218.843,363.765,-75.298,-175.918,7.641,148.276
C08086=1218.838,364.013,-75.331,-175.916,7.645,148.276
C08087=1218.834,364.260,-75.364,-175.915,7.648,148.276
C08088=1218.830,364.509,-75.397,-175.913,7.650,148.277
C08089=1218.826,364.756,-75.430,-175.912,7.653,148.277
C08090=1218.822,365.004,-75.462,-175.911,7.656,148.277
C08091=1218.818,365.252,-75.495,-175.909,7.659,148.278
C08092=1218.814,365.499,-75.529,-175.908,7.662,148.278
C08093=1218.810,365.747,-75.562,-175.906,7.665,148.278
C08094=1218.806,365.995,-75.595,-175.905,7.667,148.279
C08095=1218.802,366.243,-75.628,-175.903,7.670,148.279
C08096=1218.797,366.490,-75.661,-175.901,7.674,148.279
C08097=1218.793,366.771,-75.698,-175.900,7.676,148.280
C08098=1218.789,367.051,-75.736,-175.898,7.680,148.280
C08099=1218.784,367.330,-75.773,-175.897,7.683,148.280
C08100=1218.779,367.610,-75.811,-175.895,7.686,148.281
C08101=1218.775,367.858,-75.843,-175.894,7.689,148.281
C08102=1218.771,368.106,-75.877,-175.892,7.691,148.281
C08103=1218.767,368.353,-75.910,-175.891,7.694,148.282
C08104=1218.763,368.601,-75.944,-175.889,7.698,148.282
C08105=1218.759,368.849,-75.977,-175.888,7.700,148.282
C08106=1218.754,369.097,-76.011,-175.887,7.703,148.283
C08107=1218.750,369.344,-76.044,-175.885,7.706,148.283
C08108=1218.746,369.592,-76.077,-175.884,7.709,148.283
C08109=1218.742,369.840,-76.110,-175.883,7.711,148.284
C08110=1218.738,370.088,-76.144,-175.881,7.714,148.284
C08111=1218.734,370.336,-76.177,-175.880,7.717,148.284
C08112=1218.730,370.584,-76.210,-175.878,7.721,148.285
C08113=1218.725,370.831,-76.243,-175.877,7.723,148.285
C08114=1218.721,371.079,-76.276,-175.876,7.726,148.285
C08115=1218.717,371.327,-76.309,-175.874,7.729,148.286
C08116=1218.713,371.574,-76.343,-175.873,7.732,148.286
C08117=1218.709,371.822,-76.376,-175.872,7.735,148.287
C08118=1218.705,372.069,-76.409,-175.871,7.737,148.287
C08119=1218.701,372.317,-76.443,-175.869,7.740,148.287
C08120=1218.696,372.565,-76.476,-175.868,7.743,148.288
C08121=1218.692,372.814,-76.510,-175.867,7.746,148.288
C08122=1218.689,373.061,-76.544,-175.866,7.748,148.288
C08123=1218.685,373.308,-76.577,-175.865,7.751,148.289
C08124=1218.680,373.556,-76.610,-175.863,7.754,148.289
C08125=1218.676,373.804,-76.643,-175.862,7.757,148.290
C08126=1218.672,374.052,-76.676,-175.861,7.759,148.290
C08127=1218.668,374.299,-76.711,-175.859,7.762,148.290
C08128=1218.663,374.547,-76.744,-175.858,7.765,148.291
C08129=1218.660,374.795,-76.778,-175.857,7.768,148.291
C08130=1218.656,375.043,-76.811,-175.856,7.771,148.291
C08131=1218.652,375.290,-76.845,-175.855,7.773,148.292
C08132=1218.648,375.538,-76.878,-175.853,7.776,148.292
C08133=1218.643,375.786,-76.911,-175.852,7.779,148.293
C08134=1218.639,376.034,-76.945,-175.851,7.782,148.293
C08135=1218.635,376.281,-76.979,-175.850,7.785,148.293
C08136=1218.631,376.529,-77.012,-175.849,7.787,148.294
C08137=1218.627,376.777,-77.045,-175.848,7.790,148.294
C08138=1218.623,377.024,-77.080,-175.846,7.793,148.295
C08139=1218.619,377.272,-77.113,-175.845,7.796,148.295
C08140=1218.614,377.520,-77.146,-175.844,7.799,148.295
C08141=1218.611,377.767,-77.180,-175.843,7.802,148.296
C08142=1218.607,378.015,-77.213,-175.842,7.804,148.296
C08143=1218.602,378.263,-77.248,-175.840,7.807,148.296
C08144=1218.598,378.510,-77.281,-175.839,7.810,148.297
C08145=1218.594,378.758,-77.314,-175.838,7.813,148.297
C08146=1218.590,379.005,-77.348,-175.837,7.816,148.298
C08147=1218.585,379.253,-77.382,-175.836,7.818,148.298
C08148=1218.582,379.501,-77.416,-175.835,7.821,148.299
C08149=1218.578,379.749,-77.449,-175.834,7.824,148.299
C08150=1218.573,379.997,-77.483,-175.833,7.826,148.299
C08151=1218.569,380.244,-77.517,-175.832,7.829,148.300
C08152=1218.565,380.492,-77.550,-175.831,7.832,148.300
C08153=1218.562,380.740,-77.584,-175.830,7.835,148.301
C08154=1218.557,380.988,-77.618,-175.828,7.838,148.301
C08155=1218.553,381.235,-77.652,-175.828,7.840,148.301
C08156=1218.549,381.482,-77.685,-175.827,7.842,148.302
C08157=1218.545,381.730,-77.719,-175.826,7.846,148.302
C08158=1218.541,381.978,-77.753,-175.825,7.848,148.303
C08159=1218.537,382.225,-77.787,-175.823,7.851,148.303
C08160=1218.532,382.473,-77.821,-175.822,7.854,148.304
C08161=1218.529,382.720,-77.854,-175.822,7.856,148.304
C08162=1218.525,382.969,-77.888,-175.820,7.859,148.304
C08163=1218.520,383.216,-77.922,-175.820,7.862,148.305
C08164=1218.516,383.464,-77.956,-175.818,7.865,148.305
C08165=1218.512,383.711,-77.989,-175.817,7.868,148.306
C08166=1218.508,383.960,-78.024,-175.817,7.870,148.306
C08167=1218.504,384.207,-78.057,-175.815,7.872,148.306
C08168=1218.500,384.454,-78.092,-175.815,7.875,148.307
C08169=1218.496,384.702,-78.125,-175.814,7.878,148.307
C08170=1218.492,384.950,-78.159,-175.813,7.880,148.308
C08171=1218.488,385.198,-78.193,-175.812,7.883,148.308
C08172=1218.484,385.445,-78.227,-175.811,7.886,148.309
C08173=1218.480,385.692,-78.261,-175.810,7.889,148.309
C08174=1218.476,385.941,-78.295,-175.809,7.891,148.309
C08175=1218.472,386.188,-78.329,-175.808,7.894,148.310
C08176=1218.467,386.436,-78.363,-175.807,7.897,148.310
C08177=1218.463,386.683,-78.396,-175.806,7.900,148.311
C08178=1218.460,386.931,-78.431,-175.805,7.902,148.311
C08179=1218.455,387.179,-78.464,-175.805,7.905,148.312
C08180=1218.451,387.426,-78.498,-175.803,7.908,148.312
C08181=1218.447,387.674,-78.533,-175.803,7.910,148.312
C08182=1218.443,387.922,-78.566,-175.802,7.912,148.313
C08183=1218.438,388.169,-78.601,-175.801,7.916,148.313
C08184=1218.435,388.417,-78.635,-175.800,7.918,148.314
C08185=1218.431,388.665,-78.669,-175.799,7.920,148.314
C08186=1218.427,388.912,-78.703,-175.798,7.923,148.315
C08187=1218.423,389.160,-78.736,-175.798,7.925,148.315
C08188=1218.419,389.408,-78.771,-175.797,7.928,148.316
C08189=1218.415,389.655,-78.805,-175.796,7.931,148.316
C08190=1218.410,389.903,-78.839,-175.795,7.933,148.316
C08191=1218.407,390.151,-78.873,-175.794,7.936,148.317
C08192=1218.402,390.398,-78.908,-175.794,7.938,148.317
C08193=1218.398,390.645,-78.941,-175.793,7.941,148.318
C08194=1218.394,390.894,-78.976,-175.791,7.944,148.318
C08195=1218.390,391.141,-79.009,-175.791,7.946,148.319
C08196=1218.386,391.388,-79.044,-175.790,7.949,148.319
C08197=1218.382,391.636,-79.078,-175.790,7.951,148.320
C08198=1218.378,391.884,-79.112,-175.789,7.954,148.320
C08199=1218.374,392.131,-79.146,-175.788,7.956,148.320
C08200=1218.370,392.380,-79.181,-175.787,7.959,148.321
C08201=1218.366,392.661,-79.219,-175.786,7.962,148.321
C08202=1218.360,392.943,-79.258,-175.785,7.965,148.322
C08203=1218.356,393.225,-79.298,-175.784,7.968,148.322
C08204=1218.351,393.507,-79.336,-175.783,7.971,148.323
C08205=1218.347,393.754,-79.370,-175.783,7.973,148.323
C08206=1218.343,394.002,-79.405,-175.782,7.976,148.324
C08207=1218.339,394.249,-79.439,-175.781,7.978,148.324
C08208=1218.336,394.497,-79.473,-175.781,7.981,148.325
C08209=1218.331,394.745,-79.508,-175.780,7.983,148.325
C08210=1218.327,394.992,-79.542,-175.779,7.986,148.326
C08211=1218.323,395.240,-79.576,-175.779,7.988,148.326
C08212=1218.318,395.488,-79.610,-175.777,7.991,148.327
C08213=1218.314,395.735,-79.644,-175.777,7.994,148.327
C08214=1218.310,395.983,-79.679,-175.776,7.996,148.328
C08215=1218.307,396.230,-79.713,-175.776,7.999,148.328
C08216=1218.303,396.478,-79.748,-175.775,8.001,148.328
C08217=1218.298,396.726,-79.782,-175.774,8.004,148.329
C08218=1218.294,396.973,-79.816,-175.774,8.006,148.329
C08219=1218.290,397.221,-79.851,-175.773,8.008,148.330
C08220=1218.286,397.468,-79.885,-175.772,8.011,148.330
C08221=1218.282,397.715,-79.919,-175.771,8.014,148.331
C08222=1218.278,397.964,-79.954,-175.771,8.016,148.331
C08223=1218.274,398.211,-79.988,-175.770,8.018,148.332
C08224=1218.270,398.459,-80.023,-175.770,8.021,148.332
C08225=1218.266,398.706,-80.057,-175.769,8.023,148.332
C08226=1218.262,398.953,-80.091,-175.768,8.026,148.333
C08227=1218.258,399.201,-80.126,-175.768,8.028,148.333
C08228=1218.254,399.449,-80.160,-175.767,8.030,148.334
C08229=1218.250,399.697,-80.194,-175.766,8.033,148.334
C08230=1218.245,399.944,-80.229,-175.766,8.035,148.335
C08231=1218.242,400.191,-80.263,-175.765,8.037,148.335
C08232=1218.238,400.439,-80.298,-175.764,8.040,148.336
C08233=1218.233,400.687,-80.332,-175.764,8.042,148.336
C08234=1218.230,400.935,-80.366,-175.763,8.044,148.337
C08235=1218.225,401.182,-80.401,-175.763,8.047,148.337
C08236=1218.221,401.430,-80.436,-175.762,8.049,148.337
C08237=1218.217,401.677,-80.470,-175.762,8.052,148.338
C08238=1218.213,401.925,-80.504,-175.761,8.055,148.338
C08239=1218.209,402.173,-80.539,-175.760,8.057,148.339
C08240=1218.204,402.420,-80.573,-175.760,8.059,148.339
C08241=1218.201,402.668,-80.608,-175.759,8.062,148.340
C08242=1218.197,402.915,-80.643,-175.758,8.064,148.340
C08243=1218.193,403.163,-80.678,-175.758,8.066,148.341
C08244=1218.189,403.410,-80.711,-175.757,8.069,148.341
C08245=1218.185,403.658,-80.746,-175.757,8.071,148.342
C08246=1218.180,403.906,-80.781,-175.756,8.073,148.342
C08247=1218.177,404.153,-80.815,-175.756,8.075,148.343
C08248=1218.173,404.401,-80.849,-175.755,8.078,148.343
C08249=1218.168,404.648,-80.884,-175.755,8.081,148.344
C08250=1218.164,404.896,-80.919,-175.754,8.083,148.344
C08251=1218.161,405.143,-80.953,-175.754,8.085,148.344
C08252=1218.157,405.391,-80.988,-175.753,8.088,148.345
C08253=1218.152,405.638,-81.023,-175.752,8.090,148.345
C08254=1218.148,405.886,-81.057,-175.752,8.092,148.346
C08255=1218.144,406.134,-81.091,-175.752,8.094,148.346
C08256=1218.141,406.381,-81.127,-175.750,8.097,148.347
C08257=1218.136,406.629,-81.161,-175.750,8.099,148.347
C08258=1218.132,406.877,-81.196,-175.749,8.101,148.347
C08259=1218.128,407.124,-81.230,-175.749,8.103,148.348
C08260=1218.124,407.372,-81.265,-175.749,8.105,148.348
C08261=1218.120,407.619,-81.300,-175.748,8.109,148.349
C08262=1218.116,407.867,-81.335,-175.747,8.111,148.349
C08263=1218.112,408.114,-81.369,-175.747,8.113,148.350
C08264=1218.108,408.362,-81.404,-175.746,8.115,148.350
C08265=1218.104,408.609,-81.439,-175.746,8.117,148.351
C08266=1218.099,408.856,-81.473,-175.746,8.119,148.351
C08267=1218.095,409.104,-81.508,-175.745,8.122,148.352
C08268=1218.092,409.352,-81.542,-175.744,8.124,148.352
C08269=1218.088,409.599,-81.577,-175.744,8.126,148.353
C08270=1218.084,409.847,-81.612,-175.743,8.128,148.353
C08271=1218.079,410.094,-81.647,-175.743,8.131,148.353
C08272=1218.075,410.343,-81.682,-175.742,8.133,148.354
C08273=1218.072,410.589,-81.716,-175.742,8.135,148.354
C08274=1218.068,410.837,-81.751,-175.741,8.138,148.355
C08275=1218.063,411.085,-81.785,-175.741,8.140,148.355
C08276=1218.060,411.332,-81.821,-175.740,8.142,148.356
C08277=1218.055,411.580,-81.855,-175.740,8.144,148.356
C08278=1218.052,411.827,-81.890,-175.739,8.146,148.356
C08279=1218.048,412.074,-81.925,-175.739,8.148,148.357
C08280=1218.044,412.322,-81.960,-175.739,8.150,148.357
C08281=1218.039,412.570,-81.994,-175.738,8.152,148.358
C08282=1218.035,412.817,-82.030,-175.738,8.155,148.358
C08283=1218.031,413.065,-82.064,-175.737,8.157,148.359
C08284=1218.027,413.313,-82.099,-175.736,8.160,148.359
C08285=1218.023,413.559,-82.134,-175.736,8.162,148.359
C08286=1218.019,413.807,-82.168,-175.735,8.164,148.360
C08287=1218.015,414.055,-82.203,-175.735,8.166,148.360
C08288=1218.011,414.302,-82.238,-175.735,8.168,148.361
C08289=1218.007,414.550,-82.273,-175.734,8.170,148.361
C08290=1218.003,414.798,-82.308,-175.734,8.172,148.362
C08291=1217.999,415.045,-82.343,-175.733,8.174,148.362
C08292=1217.995,415.292,-82.377,-175.733,8.177,148.363
C08293=1217.991,415.517,-82.409,-175.732,8.179,148.363
C08294=1217.988,415.742,-82.441,-175.732,8.181,148.363
C08295=1217.984,415.966,-82.473,-175.731,8.183,148.364
C08296=1217.981,416.192,-82.504,-175.731,8.185,148.364
C08297=1217.977,416.416,-82.536,-175.731,8.186,148.364
C08298=1217.972,416.641,-82.568,-175.730,8.188,148.365
C08299=1217.970,416.865,-82.599,-175.730,8.190,148.365
C08300=1217.971,417.090,-82.631,-175.729,8.192,148.366
C08301=1217.549,417.090,-82.666,-175.733,8.203,148.369
C08302=1217.548,416.864,-82.634,-175.733,8.201,148.369
C08303=1217.551,416.638,-82.602,-175.733,8.199,148.368
C08304=1217.555,416.412,-82.570,-175.734,8.197,148.368
C08305=1217.559,416.187,-82.538,-175.734,8.196,148.368
C08306=1217.562,415.960,-82.506,-175.734,8.193,148.367
C08307=1217.566,415.734,-82.475,-175.735,8.191,148.367
C08308=1217.569,415.508,-82.443,-175.736,8.189,148.367
C08309=1217.573,415.282,-82.411,-175.736,8.187,148.366
C08310=1217.577,415.034,-82.377,-175.737,8.185,148.366
C08311=1217.581,414.787,-82.341,-175.737,8.183,148.365
C08312=1217.585,414.539,-82.306,-175.737,8.181,148.365
C08313=1217.589,414.292,-82.271,-175.738,8.179,148.364
C08314=1217.593,414.044,-82.236,-175.738,8.177,148.364
C08315=1217.597,413.797,-82.202,-175.738,8.174,148.364
C08316=1217.601,413.549,-82.167,-175.739,8.172,148.363
C08317=1217.605,413.302,-82.132,-175.739,8.170,148.363
C08318=1217.609,413.054,-82.098,-175.740,8.168,148.362
C08319=1217.614,412.807,-82.062,-175.741,8.165,148.362
C08320=1217.618,412.559,-82.028,-175.741,8.163,148.361
C08321=1217.622,412.311,-81.993,-175.742,8.161,148.361
C08322=1217.625,412.064,-81.958,-175.742,8.159,148.360
C08323=1217.630,411.817,-81.924,-175.742,8.157,148.360
C08324=1217.634,411.569,-81.889,-175.743,8.155,148.360
C08325=1217.637,411.321,-81.853,-175.744,8.153,148.359
C08326=1217.642,411.074,-81.819,-175.744,8.150,148.359
C08327=1217.646,410.826,-81.784,-175.745,8.148,148.358
C08328=1217.649,410.579,-81.749,-175.745,8.145,148.358
C08329=1217.653,410.331,-81.715,-175.746,8.143,148.357
C08330=1217.658,410.084,-81.680,-175.746,8.141,148.357
C08331=1217.662,409.836,-81.645,-175.747,8.139,148.357
C08332=1217.666,409.589,-81.610,-175.747,8.137,148.356
C08333=1217.669,409.341,-81.576,-175.748,8.135,148.356
C08334=1217.674,409.094,-81.541,-175.748,8.132,148.355
C08335=1217.678,408.846,-81.506,-175.749,8.130,148.355
C08336=1217.682,408.599,-81.471,-175.749,8.127,148.354
C08337=1217.686,408.350,-81.437,-175.750,8.125,148.354
C08338=1217.690,408.103,-81.403,-175.750,8.123,148.353
C08339=1217.694,407.856,-81.367,-175.751,8.121,148.353
C08340=1217.698,407.608,-81.333,-175.751,8.119,148.353
C08341=1217.702,407.360,-81.298,-175.752,8.116,148.352
C08342=1217.706,407.113,-81.264,-175.752,8.114,148.352
C08343=1217.710,406.865,-81.229,-175.753,8.112,148.351
C08344=1217.714,406.618,-81.194,-175.753,8.110,148.351
C08345=1217.718,406.370,-81.159,-175.754,8.108,148.350
C08346=1217.722,406.123,-81.125,-175.755,8.104,148.350
C08347=1217.727,405.876,-81.091,-175.755,8.103,148.349
C08348=1217.731,405.628,-81.056,-175.755,8.100,148.349
C08349=1217.735,405.381,-81.021,-175.756,8.098,148.348
C08350=1217.738,405.133,-80.987,-175.757,8.095,148.348
C08351=1217.743,404.886,-80.952,-175.757,8.093,148.347
C08352=1217.747,404.637,-80.917,-175.758,8.091,148.347
C08353=1217.751,404.390,-80.883,-175.758,8.089,148.347
C08354=1217.754,404.142,-80.849,-175.759,8.086,148.346
C08355=1217.759,403.895,-80.813,-175.759,8.084,148.346
C08356=1217.763,403.647,-80.779,-175.760,8.082,148.345
C08357=1217.767,403.400,-80.744,-175.760,8.079,148.345
C08358=1217.770,403.152,-80.710,-175.761,8.077,148.344
C08359=1217.775,402.905,-80.675,-175.761,8.074,148.344
C08360=1217.780,402.657,-80.641,-175.762,8.072,148.343
C08361=1217.783,402.409,-80.607,-175.763,8.069,148.343
C08362=1217.787,402.162,-80.572,-175.763,8.067,148.343
C08363=1217.791,401.914,-80.537,-175.764,8.065,148.342
C08364=1217.795,401.667,-80.503,-175.764,8.063,148.342
C08365=1217.799,401.419,-80.468,-175.765,8.060,148.341
C08366=1217.803,401.172,-80.433,-175.766,8.058,148.341
C08367=1217.808,400.924,-80.399,-175.766,8.056,148.340
C08368=1217.811,400.677,-80.365,-175.767,8.053,148.340
C08369=1217.816,400.429,-80.330,-175.768,8.051,148.339
C08370=1217.820,400.181,-80.295,-175.768,8.049,148.339
C08371=1217.824,399.934,-80.262,-175.769,8.046,148.338
C08372=1217.828,399.686,-80.227,-175.769,8.043,148.338
C08373=1217.832,399.438,-80.192,-175.770,8.041,148.338
C08374=1217.836,399.191,-80.158,-175.771,8.038,148.337
C08375=1217.840,398.943,-80.124,-175.771,8.036,148.337
C08376=1217.844,398.696,-80.090,-175.772,8.033,148.336
C08377=1217.848,398.448,-80.055,-175.773,8.031,148.336
C08378=1217.852,398.200,-80.020,-175.773,8.028,148.335
C08379=1217.856,397.953,-79.987,-175.774,8.026,148.335
C08380=1217.860,397.705,-79.952,-175.774,8.024,148.334
C08381=1217.865,397.458,-79.917,-175.775,8.021,148.334
C08382=1217.868,397.210,-79.883,-175.776,8.019,148.333
C08383=1217.872,396.963,-79.849,-175.777,8.016,148.333
C08384=1217.876,396.716,-79.815,-175.777,8.014,148.333
C08385=1217.880,396.467,-79.780,-175.778,8.012,148.332
C08386=1217.885,396.220,-79.745,-175.779,8.009,148.332
C08387=1217.888,395.972,-79.711,-175.779,8.007,148.331
C08388=1217.893,395.725,-79.677,-175.780,8.004,148.331
C08389=1217.896,395.478,-79.643,-175.780,8.002,148.330
C08390=1217.900,395.229,-79.608,-175.782,7.999,148.330
C08391=1217.905,394.981,-79.574,-175.782,7.997,148.329
C08392=1217.909,394.734,-79.540,-175.783,7.994,148.329
C08393=1217.913,394.486,-79.506,-175.784,7.992,148.328
C08394=1217.917,394.239,-79.472,-175.784,7.989,148.328
C08395=1217.921,393.991,-79.437,-175.785,7.987,148.328
C08396=1217.925,393.744,-79.403,-175.786,7.984,148.327
C08397=1217.929,393.496,-79.368,-175.786,7.982,148.327
C08398=1217.935,393.214,-79.330,-175.787,7.978,148.326
C08399=1217.938,392.932,-79.291,-175.788,7.976,148.326
C08400=1217.943,392.650,-79.252,-175.789,7.972,148.325
C08401=1217.947,392.369,-79.213,-175.790,7.969,148.324
C08402=1217.952,392.121,-79.178,-175.790,7.967,148.324
C08403=1217.955,391.873,-79.144,-175.792,7.965,148.324
C08404=1217.960,391.625,-79.110,-175.792,7.961,148.323
C08405=1217.964,391.378,-79.077,-175.793,7.960,148.323
C08406=1217.968,391.130,-79.042,-175.794,7.957,148.322
C08407=1217.972,390.883,-79.008,-175.794,7.954,148.322
C08408=1217.976,390.636,-78.973,-175.796,7.952,148.321
C08409=1217.980,390.387,-78.940,-175.796,7.948,148.321
C08410=1217.984,390.140,-78.905,-175.797,7.947,148.320
C08411=1217.988,389.893,-78.872,-175.798,7.944,148.320
C08412=1217.992,389.644,-78.837,-175.798,7.941,148.320
C08413=1217.996,389.397,-78.804,-175.800,7.939,148.319
C08414=1218.001,389.149,-78.769,-175.801,7.936,148.319
C08415=1218.004,388.902,-78.735,-175.801,7.934,148.318
C08416=1218.009,388.654,-78.700,-175.802,7.931,148.318
C08417=1218.013,388.406,-78.667,-175.803,7.928,148.317
C08418=1218.017,388.159,-78.633,-175.803,7.926,148.317
C08419=1218.021,387.911,-78.599,-175.805,7.923,148.316
C08420=1218.025,387.663,-78.565,-175.806,7.920,148.316
C08421=1218.029,387.416,-78.531,-175.806,7.918,148.316
C08422=1218.033,387.168,-78.497,-175.807,7.915,148.315
C08423=1218.037,386.921,-78.462,-175.808,7.912,148.315
C08424=1218.041,386.673,-78.429,-175.809,7.910,148.314
C08425=1218.046,386.426,-78.395,-175.810,7.907,148.314
C08426=1218.049,386.177,-78.361,-175.811,7.904,148.313
C08427=1218.054,385.930,-78.327,-175.812,7.901,148.313
C08428=1218.058,385.683,-78.293,-175.812,7.899,148.312
C08429=1218.061,385.434,-78.259,-175.814,7.896,148.312
C08430=1218.066,385.187,-78.225,-175.815,7.893,148.312
C08431=1218.070,384.940,-78.191,-175.816,7.891,148.311
C08432=1218.075,384.692,-78.157,-175.816,7.888,148.311
C08433=1218.078,384.444,-78.123,-175.817,7.886,148.310
C08434=1218.082,384.196,-78.090,-175.819,7.883,148.310
C08435=1218.087,383.949,-78.055,-175.820,7.880,148.310
C08436=1218.090,383.702,-78.021,-175.820,7.878,148.309
C08437=1218.094,383.453,-77.988,-175.821,7.875,148.309
C08438=1218.098,383.206,-77.953,-175.822,7.872,148.308
C08439=1218.103,382.958,-77.920,-175.823,7.869,148.308
C08440=1218.106,382.711,-77.886,-175.825,7.866,148.307
C08441=1218.111,382.462,-77.852,-175.825,7.864,148.307
C08442=1218.115,382.215,-77.818,-175.826,7.861,148.306
C08443=1218.119,381.967,-77.785,-175.827,7.858,148.306
C08444=1218.123,381.720,-77.751,-175.828,7.856,148.306
C08445=1218.127,381.472,-77.718,-175.830,7.853,148.305
C08446=1218.131,381.224,-77.683,-175.831,7.850,148.305
C08447=1218.135,380.976,-77.650,-175.831,7.848,148.305
C08448=1218.139,380.729,-77.616,-175.832,7.845,148.304
C08449=1218.143,380.481,-77.583,-175.833,7.842,148.304
C08450=1218.148,380.234,-77.548,-175.835,7.839,148.303
C08451=1218.152,379.986,-77.515,-175.836,7.836,148.303
C08452=1218.155,379.739,-77.481,-175.837,7.834,148.302
C08453=1218.160,379.490,-77.447,-175.838,7.831,148.302
C08454=1218.164,379.243,-77.413,-175.839,7.828,148.302
C08455=1218.168,378.996,-77.380,-175.840,7.826,148.301
C08456=1218.172,378.747,-77.346,-175.841,7.823,148.301
C08457=1218.176,378.500,-77.312,-175.842,7.820,148.300
C08458=1218.180,378.252,-77.279,-175.843,7.817,148.300
C08459=1218.184,378.005,-77.245,-175.844,7.814,148.299
C08460=1218.188,377.757,-77.212,-175.845,7.812,148.299
C08461=1218.193,377.508,-77.178,-175.847,7.809,148.299
C08462=1218.197,377.261,-77.144,-175.848,7.806,148.298
C08463=1218.201,377.014,-77.111,-175.849,7.803,148.298
C08464=1218.205,376.766,-77.077,-175.850,7.800,148.297
C08465=1218.209,376.519,-77.043,-175.851,7.798,148.297
C08466=1218.214,376.271,-77.010,-175.852,7.795,148.297
C08467=1218.218,376.023,-76.977,-175.854,7.792,148.296
C08468=1218.221,375.775,-76.942,-175.855,7.789,148.296
C08469=1218.225,375.528,-76.909,-175.856,7.786,148.296
C08470=1218.229,375.280,-76.876,-175.857,7.783,148.295
C08471=1218.234,375.032,-76.842,-175.858,7.781,148.295
C08472=1218.238,374.785,-76.809,-175.860,7.778,148.294
C08473=1218.242,374.537,-76.775,-175.861,7.775,148.294
C08474=1218.246,374.289,-76.742,-175.862,7.773,148.294
C08475=1218.250,374.041,-76.709,-175.864,7.770,148.293
C08476=1218.254,373.794,-76.675,-175.865,7.767,148.293
C08477=1218.258,373.546,-76.641,-175.866,7.764,148.293
C08478=1218.263,373.298,-76.608,-175.867,7.761,148.292
C08479=1218.267,373.050,-76.575,-175.868,7.758,148.292
C08480=1218.271,372.803,-76.541,-175.870,7.756,148.291
C08481=1218.275,372.555,-76.508,-175.871,7.753,148.291
C08482=1218.279,372.308,-76.475,-175.872,7.750,148.291
C08483=1218.282,372.059,-76.441,-175.874,7.747,148.290
C08484=1218.286,371.811,-76.408,-175.875,7.745,148.290
C08485=1218.291,371.563,-76.374,-175.876,7.742,148.290
C08486=1218.295,371.316,-76.340,-175.877,7.739,148.289
C08487=1218.299,371.069,-76.307,-175.878,7.736,148.289
C08488=1218.303,370.821,-76.274,-175.880,7.733,148.289
C08489=1218.308,370.573,-76.241,-175.882,7.730,148.288
C08490=1218.312,370.325,-76.208,-175.883,7.727,148.288
C08491=1218.316,370.078,-76.175,-175.884,7.724,148.287
C08492=1218.320,369.830,-76.141,-175.885,7.722,148.287
C08493=1218.324,369.582,-76.108,-175.887,7.719,148.287
C08494=1218.328,369.334,-76.075,-175.888,7.716,148.286
C08495=1218.332,369.087,-76.042,-175.889,7.713,148.286
C08496=1218.336,368.838,-76.008,-175.891,7.710,148.286
C08497=1218.340,368.591,-75.974,-175.893,7.707,148.285
C08498=1218.344,368.343,-75.941,-175.894,7.704,148.285
C08499=1218.348,368.096,-75.908,-175.895,7.702,148.285
C08500=1218.352,367.848,-75.875,-175.897,7.699,148.284
C08501=1218.356,367.600,-75.842,-175.898,7.696,148.284
C08502=1218.362,367.320,-75.804,-175.900,7.693,148.284
C08503=1218.367,367.040,-75.767,-175.901,7.689,148.283
C08504=1218.371,366.761,-75.729,-175.903,7.686,148.283
C08505=1218.375,366.480,-75.692,-175.905,7.683,148.283
C08506=1218.380,366.232,-75.659,-175.906,7.680,148.282
C08507=1218.384,365.984,-75.626,-175.907,7.677,148.282
C08508=1218.388,365.736,-75.593,-175.909,7.675,148.282
C08509=1218.392,365.489,-75.560,-175.911,7.671,148.281
C08510=1218.396,365.241,-75.526,-175.912,7.668,148.281
C08511=1218.400,364.993,-75.493,-175.913,7.666,148.281
C08512=1218.404,364.746,-75.461,-175.915,7.663,148.280
C08513=1218.408,364.498,-75.428,-175.916,7.660,148.280
C08514=1218.412,364.250,-75.394,-175.918,7.657,148.280
C08515=1218.416,364.002,-75.362,-175.919,7.654,148.279
C08516=1218.421,363.754,-75.329,-175.921,7.652,148.279
C08517=1218.425,363.507,-75.296,-175.922,7.649,148.279
C08518=1218.429,363.259,-75.262,-175.924,7.645,148.278
C08519=1218.433,363.011,-75.229,-175.926,7.643,148.278
C08520=1218.437,362.763,-75.196,-175.927,7.640,148.278
C08521=1218.442,362.515,-75.164,-175.928,7.637,148.278
C08522=1218.446,362.268,-75.132,-175.931,7.634,148.277
C08523=1218.450,362.021,-75.098,-175.932,7.631,148.277
C08524=1218.454,361.773,-75.065,-175.933,7.629,148.277
C08525=1218.458,361.525,-75.032,-175.935,7.626,148.276
C08526=1218.462,361.277,-75.000,-175.937,7.622,148.276
C08527=1218.467,361.029,-74.966,-175.938,7.620,148.276
C08528=1218.470,360.782,-74.934,-175.940,7.617,148.276
C08529=1218.474,360.534,-74.901,-175.941,7.614,148.275
C08530=1218.479,360.286,-74.868,-175.943,7.611,148.275
C08531=1218.483,360.038,-74.835,-175.945,7.608,148.275
C08532=1218.487,359.790,-74.802,-175.946,7.605,148.274
C08533=1218.491,359.542,-74.770,-175.948,7.602,148.274
C08534=1218.495,359.294,-74.737,-175.950,7.600,148.274
C08535=1218.499,359.047,-74.704,-175.951,7.597,148.273
C08536=1218.503,358.798,-74.671,-175.953,7.593,148.273
C08537=1218.508,358.551,-74.639,-175.954,7.591,148.273
C08538=1218.511,358.304,-74.606,-175.956,7.588,148.273
C08539=1218.516,358.055,-74.574,-175.958,7.585,148.272
C08540=1218.520,357.808,-74.540,-175.959,7.582,148.272
C08541=1218.524,357.559,-74.508,-175.961,7.579,148.272
C08542=1218.528,357.312,-74.475,-175.963,7.577,148.272
C08543=1218.532,357.064,-74.442,-175.965,7.574,148.271
C08544=1218.536,356.816,-74.410,-175.966,7.571,148.271
C08545=1218.541,356.568,-74.377,-175.968,7.568,148.271
C08546=1218.545,356.321,-74.345,-175.970,7.565,148.271
C08547=1218.549,356.073,-74.312,-175.971,7.562,148.270
C08548=1218.553,355.825,-74.280,-175.973,7.559,148.270
C08549=1218.557,355.577,-74.247,-175.975,7.556,148.270
C08550=1218.561,355.329,-74.215,-175.976,7.554,148.270
C08551=1218.565,355.081,-74.181,-175.978,7.551,148.269
C08552=1218.569,354.833,-74.150,-175.980,7.547,148.269
C08553=1218.574,354.586,-74.117,-175.981,7.545,148.269
C08554=1218.578,354.338,-74.084,-175.983,7.542,148.269
C08555=1218.582,354.090,-74.052,-175.985,7.539,148.268
C08556=1218.586,353.842,-74.019,-175.987,7.537,148.268
C08557=1218.590,353.594,-73.986,-175.988,7.534,148.268
C08558=1218.594,353.346,-73.954,-175.990,7.530,148.268
C08559=1218.599,353.099,-73.922,-175.992,7.528,148.267
C08560=1218.603,352.851,-73.889,-175.994,7.524,148.267
C08561=1218.607,352.603,-73.857,-175.996,7.522,148.267
C08562=1218.611,352.355,-73.825,-175.997,7.519,148.267
C08563=1218.615,352.107,-73.792,-176.000,7.516,148.267
C08564=1218.620,351.859,-73.760,-176.001,7.513,148.266
C08565=1218.624,351.612,-73.727,-176.002,7.511,148.266
C08566=1218.628,351.364,-73.695,-176.005,7.507,148.266
C08567=1218.632,351.115,-73.663,-176.006,7.505,148.266
C08568=1218.635,350.868,-73.630,-176.008,7.502,148.265
C08569=1218.641,350.620,-73.598,-176.010,7.499,148.265
C08570=1218.644,350.372,-73.566,-176.012,7.496,148.265
C08571=1218.649,350.124,-73.534,-176.014,7.493,148.265
C08572=1218.653,349.876,-73.501,-176.015,7.491,148.265
C08573=1218.657,349.629,-73.469,-176.017,7.488,148.264
C08574=1218.662,349.380,-73.437,-176.019,7.485,148.264
C08575=1218.665,349.132,-73.405,-176.021,7.482,148.264
C08576=1218.669,348.885,-73.372,-176.023,7.480,148.264
C08577=1218.674,348.637,-73.340,-176.025,7.476,148.264
C08578=1218.678,348.389,-73.308,-176.026,7.474,148.263
C08579=1218.682,348.141,-73.276,-176.029,7.470,148.263
C08580=1218.686,347.893,-73.244,-176.030,7.468,148.263
C08581=1218.690,347.646,-73.211,-176.032,7.465,148.263
C08582=1218.695,347.398,-73.179,-176.034,7.462,148.263
C08583=1218.698,347.150,-73.147,-176.036,7.459,148.262
C08584=1218.703,346.902,-73.115,-176.038,7.456,148.262
C08585=1218.707,346.654,-73.083,-176.040,7.454,148.262
C08586=1218.711,346.406,-73.051,-176.041,7.451,148.262
C08587=1218.715,346.157,-73.019,-176.043,7.448,148.262
C08588=1218.720,345.910,-72.987,-176.045,7.445,148.261
C08589=1218.724,345.662,-72.954,-176.047,7.442,148.261
C08590=1218.727,345.414,-72.922,-176.049,7.439,148.261
C08591=1218.733,345.167,-72.890,-176.051,7.437,148.261
C08592=1218.736,344.919,-72.859,-176.053,7.433,148.261
C08593=1218.740,344.671,-72.827,-176.054,7.431,148.260
C08594=1218.745,344.423,-72.795,-176.057,7.428,148.260
C08595=1218.749,344.175,-72.763,-176.059,7.425,148.260
C08596=1218.753,343.927,-72.730,-176.060,7.423,148.260
C08597=1218.757,343.679,-72.699,-176.062,7.419,148.260
C08598=1218.761,343.431,-72.667,-176.064,7.417,148.260
C08599=1218.766,343.183,-72.635,-176.066,7.414,148.259
C08600=1218.770,342.936,-72.603,-176.068,7.411,148.259
C08601=1218.774,342.687,-72.571,-176.070,7.409,148.259
C08602=1218.779,342.440,-72.539,-176.072,7.405,148.259
C08603=1218.782,342.192,-72.507,-176.074,7.403,148.259
C08604=1218.786,341.943,-72.476,-176.076,7.400,148.259
C08605=1218.791,341.695,-72.444,-176.078,7.397,148.258
C08606=1218.796,341.418,-72.409,-176.080,7.394,148.258
C08607=1218.801,341.140,-72.372,-176.083,7.391,148.258
C08608=1218.805,340.862,-72.337,-176.085,7.387,148.258
C08609=1218.810,340.584,-72.302,-176.086,7.385,148.258
C08610=1218.814,340.336,-72.269,-176.089,7.381,148.258
C08611=1218.818,340.088,-72.238,-176.090,7.379,148.257
C08612=1218.822,339.841,-72.206,-176.093,7.376,148.257
C08613=1218.826,339.592,-72.175,-176.095,7.373,148.257
C08614=1218.831,339.344,-72.143,-176.096,7.371,148.257
C08615=1218.835,339.096,-72.111,-176.098,7.367,148.257
C08616=1218.839,338.848,-72.079,-176.100,7.365,148.257
C08617=1218.843,338.601,-72.048,-176.103,7.362,148.257
C08618=1218.848,338.352,-72.016,-176.104,7.359,148.256
C08619=1218.852,338.105,-71.984,-176.107,7.356,148.256
C08620=1218.856,337.857,-71.953,-176.109,7.354,148.256
C08621=1218.860,337.609,-71.921,-176.110,7.351,148.256
C08622=1218.864,337.361,-71.890,-176.113,7.348,148.256
C08623=1218.869,337.112,-71.858,-176.115,7.346,148.256
C08624=1218.873,336.865,-71.826,-176.117,7.342,148.256
C08625=1218.877,336.616,-71.795,-176.118,7.340,148.256
C08626=1218.881,336.369,-71.763,-176.121,7.337,148.256
C08627=1218.885,336.121,-71.732,-176.123,7.334,148.255
C08628=1218.889,335.873,-71.701,-176.125,7.332,148.255
C08629=1218.893,335.625,-71.669,-176.127,7.329,148.255
C08630=1218.898,335.377,-71.637,-176.129,7.326,148.255
C08631=1218.902,335.129,-71.606,-176.131,7.323,148.255
C08632=1218.907,334.881,-71.574,-176.133,7.321,148.255
C08633=1218.911,334.633,-71.543,-176.135,7.317,148.255
C08634=1218.915,334.385,-71.512,-176.137,7.315,148.255
C08635=1218.919,334.137,-71.481,-176.139,7.312,148.254
C08636=1218.923,333.889,-71.449,-176.141,7.309,148.254
C08637=1218.927,333.641,-71.417,-176.143,7.307,148.254
C08638=1218.931,333.393,-71.387,-176.145,7.304,148.254
C08639=1218.935,333.145,-71.355,-176.147,7.301,148.254
C08640=1218.940,332.897,-71.324,-176.150,7.298,148.254
C08641=1218.944,332.649,-71.292,-176.152,7.296,148.254
C08642=1218.949,332.401,-71.261,-176.154,7.292,148.254
C08643=1218.953,332.153,-71.229,-176.156,7.290,148.254
C08644=1218.957,331.905,-71.198,-176.158,7.288,148.254
C08645=1218.961,331.656,-71.167,-176.160,7.284,148.253
C08646=1218.966,331.409,-71.135,-176.162,7.282,148.253
C08647=1218.970,331.161,-71.105,-176.164,7.279,148.253
C08648=1218.974,330.913,-71.073,-176.166,7.277,148.253
C08649=1218.978,330.665,-71.042,-176.168,7.273,148.253
C08650=1218.982,330.417,-71.010,-176.171,7.271,148.253
C08651=1218.987,330.169,-70.979,-176.173,7.268,148.253
C08652=1218.991,329.920,-70.948,-176.175,7.265,148.253
C08653=1218.995,329.673,-70.917,-176.176,7.263,148.253
C08654=1218.999,329.425,-70.887,-176.179,7.260,148.253
C08655=1219.003,329.177,-70.856,-176.181,7.257,148.252
C08656=1219.007,328.929,-70.824,-176.183,7.254,148.252
C08657=1219.011,328.681,-70.793,-176.185,7.252,148.252
C08658=1219.016,328.433,-70.762,-176.188,7.249,148.252
C08659=1219.020,328.185,-70.731,-176.189,7.246,148.252
C08660=1219.024,327.937,-70.700,-176.192,7.243,148.252
C08661=1219.029,327.689,-70.669,-176.194,7.241,148.252
C08662=1219.033,327.440,-70.638,-176.196,7.238,148.252
C08663=1219.037,327.193,-70.606,-176.198,7.235,148.252
C08664=1219.042,326.945,-70.575,-176.200,7.233,148.252
C08665=1219.046,326.696,-70.544,-176.203,7.230,148.252
C08666=1219.050,326.449,-70.514,-176.204,7.227,148.252
C08667=1219.054,326.201,-70.483,-176.207,7.224,148.252
C08668=1219.058,325.953,-70.452,-176.209,7.222,148.252
C08669=1219.063,325.705,-70.421,-176.211,7.219,148.251
C08670=1219.067,325.456,-70.390,-176.213,7.216,148.251
C08671=1219.071,325.208,-70.359,-176.215,7.214,148.251
C08672=1219.075,324.960,-70.329,-176.218,7.211,148.251
C08673=1219.079,324.712,-70.297,-176.220,7.209,148.251
C08674=1219.083,324.464,-70.266,-176.222,7.205,148.251
C08675=1219.088,324.216,-70.235,-176.224,7.203,148.251
C08676=1219.092,323.968,-70.204,-176.227,7.200,148.251
C08677=1219.096,323.720,-70.174,-176.228,7.197,148.251
C08678=1219.101,323.472,-70.143,-176.231,7.194,148.251
C08679=1219.105,323.223,-70.112,-176.233,7.192,148.251
C08680=1219.109,322.975,-70.081,-176.235,7.189,148.251
C08681=1219.113,322.728,-70.051,-176.238,7.187,148.251
C08682=1219.118,322.480,-70.020,-176.240,7.184,148.251
C08683=1219.122,322.231,-69.989,-176.242,7.181,148.251
C08684=1219.126,321.983,-69.959,-176.244,7.179,148.251
C08685=1219.130,321.736,-69.928,-176.247,7.176,148.251
C08686=1219.134,321.487,-69.897,-176.248,7.173,148.251
C08687=1219.139,321.239,-69.867,-176.251,7.170,148.251
C08688=1219.143,320.991,-69.836,-176.253,7.168,148.251
C08689=1219.147,320.743,-69.806,-176.255,7.165,148.250
C08690=1219.151,320.495,-69.774,-176.257,7.162,148.250
C08691=1219.155,320.247,-69.744,-176.259,7.160,148.250
C08692=1219.160,319.999,-69.714,-176.262,7.157,148.250
C08693=1219.164,319.751,-69.683,-176.264,7.155,148.250
C08694=1219.168,319.503,-69.652,-176.266,7.152,148.250
C08695=1219.172,319.255,-69.621,-176.269,7.149,148.250
C08696=1219.177,319.006,-69.591,-176.271,7.146,148.250
C08697=1219.181,318.759,-69.561,-176.273,7.144,148.250
C08698=1219.185,318.510,-69.530,-176.275,7.142,148.250
C08699=1219.190,318.262,-69.499,-176.278,7.139,148.250
C08700=1219.194,318.014,-69.469,-176.280,7.136,148.250
C08701=1219.198,317.766,-69.438,-176.282,7.133,148.250
C08702=1219.202,317.518,-69.409,-176.284,7.131,148.250
C08703=1219.206,317.269,-69.378,-176.287,7.128,148.250
C08704=1219.211,317.022,-69.347,-176.289,7.125,148.250
C08705=1219.215,316.774,-69.317,-176.291,7.122,148.250
C08706=1219.220,316.525,-69.287,-176.293,7.120,148.250
C08707=1219.224,316.278,-69.257,-176.295,7.118,148.250
C08708=1219.228,316.029,-69.226,-176.298,7.115,148.250
C08709=1219.232,315.781,-69.195,-176.300,7.112,148.250
C08710=1219.237,315.505,-69.162,-176.303,7.109,148.250
C08711=1219.241,315.229,-69.128,-176.305,7.106,148.250
C08712=1219.246,314.954,-69.095,-176.308,7.103,148.250
C08713=1219.251,314.678,-69.061,-176.311,7.100,148.250
C08714=1219.255,314.429,-69.030,-176.312,7.098,148.250
C08715=1219.259,314.181,-69.000,-176.314,7.095,148.250
C08716=1219.264,313.933,-68.969,-176.317,7.092,148.250
C08717=1219.268,313.685,-68.940,-176.319,7.090,148.250
C08718=1219.272,313.437,-68.910,-176.322,7.087,148.250
C08719=1219.277,313.189,-68.880,-176.324,7.085,148.250
C08720=1219.281,312.941,-68.849,-176.327,7.082,148.250
C08721=1219.285,312.693,-68.819,-176.328,7.079,148.250
C08722=1219.289,312.444,-68.789,-176.331,7.076,148.250
C08723=1219.294,312.196,-68.758,-176.333,7.074,148.250
C08724=1219.298,311.948,-68.729,-176.335,7.072,148.250
C08725=1219.302,311.700,-68.698,-176.338,7.069,148.250
C08726=1219.307,311.452,-68.668,-176.340,7.067,148.250
C08727=1219.310,311.204,-68.638,-176.343,7.064,148.250
C08728=1219.315,310.955,-68.608,-176.345,7.061,148.250
C08729=1219.319,310.708,-68.578,-176.347,7.058,148.250
C08730=1219.324,310.459,-68.548,-176.349,7.056,148.250
C08731=1219.328,310.211,-68.518,-176.351,7.054,148.250
C08732=1219.332,309.963,-68.488,-176.354,7.051,148.250
C08733=1219.337,309.715,-68.458,-176.356,7.048,148.250
C08734=1219.340,309.466,-68.428,-176.359,7.045,148.250
C08735=1219.345,309.218,-68.398,-176.361,7.043,148.250
C08736=1219.349,308.970,-68.368,-176.363,7.041,148.250
C08737=1219.353,308.722,-68.338,-176.365,7.038,148.250
C08738=1219.357,308.474,-68.308,-176.368,7.036,148.250
C08739=1219.362,308.226,-68.278,-176.370,7.033,148.250
C08740=1219.366,307.977,-68.248,-176.372,7.030,148.250
C08741=1219.370,307.730,-68.218,-176.375,7.027,148.250
C08742=1219.375,307.481,-68.188,-176.377,7.025,148.250
C08743=1219.379,307.233,-68.159,-176.379,7.023,148.250
C08744=1219.384,306.985,-68.129,-176.382,7.020,148.250
C08745=1219.388,306.737,-68.099,-176.384,7.018,148.250
C08746=1219.392,306.488,-68.069,-176.387,7.015,148.250
C08747=1219.396,306.240,-68.040,-176.389,7.012,148.251
C08748=1219.400,305.992,-68.010,-176.391,7.010,148.251
C08749=1219.405,305.744,-67.979,-176.394,7.007,148.251
C08750=1219.409,305.496,-67.950,-176.396,7.005,148.251
C08751=1219.414,305.247,-67.921,-176.398,7.002,148.251
C08752=1219.418,304.999,-67.891,-176.400,7.000,148.251
C08753=1219.422,304.751,-67.861,-176.403,6.997,148.251
C08754=1219.427,304.503,-67.831,-176.405,6.994,148.251
C08755=1219.431,304.255,-67.801,-176.407,6.992,148.251
C08756=1219.435,304.006,-67.772,-176.410,6.989,148.251
C08757=1219.439,303.758,-67.743,-176.412,6.987,148.251
C08758=1219.444,303.510,-67.713,-176.415,6.984,148.251
C08759=1219.449,303.262,-67.683,-176.417,6.982,148.251
C08760=1219.453,303.014,-67.653,-176.419,6.979,148.251
C08761=1219.457,302.766,-67.624,-176.422,6.976,148.251
C08762=1219.461,302.518,-67.594,-176.424,6.974,148.251
C08763=1219.465,302.269,-67.565,-176.427,6.971,148.251
C08764=1219.469,302.021,-67.535,-176.429,6.969,148.251
C08765=1219.474,301.773,-67.506,-176.431,6.967,148.251
C08766=1219.479,301.524,-67.476,-176.434,6.964,148.251
C08767=1219.483,301.276,-67.446,-176.436,6.962,148.252
C08768=1219.487,301.028,-67.417,-176.439,6.959,148.252
C08769=1219.491,300.779,-67.388,-176.441,6.957,148.252
C08770=1219.495,300.531,-67.358,-176.443,6.954,148.252
C08771=1219.500,300.284,-67.329,-176.446,6.951,148.252
C08772=1219.504,300.035,-67.300,-176.448,6.949,148.252
C08773=1219.508,299.787,-67.270,-176.450,6.946,148.252
C08774=1219.513,299.539,-67.241,-176.452,6.944,148.252
C08775=1219.517,299.291,-67.211,-176.455,6.942,148.252
C08776=1219.521,299.042,-67.182,-176.458,6.939,148.252
C08777=1219.525,298.794,-67.152,-176.460,6.937,148.252
C08778=1219.530,298.546,-67.123,-176.462,6.934,148.252
C08779=1219.534,298.298,-67.094,-176.465,6.931,148.252
C08780=1219.539,298.049,-67.065,-176.467,6.929,148.252
C08781=1219.543,297.801,-67.036,-176.469,6.926,148.252
C08782=1219.547,297.553,-67.006,-176.472,6.924,148.252
C08783=1219.551,297.305,-66.977,-176.474,6.922,148.253
C08784=1219.555,297.056,-66.947,-176.477,6.919,148.253
C08785=1219.560,296.809,-66.918,-176.479,6.917,148.253
C08786=1219.564,296.560,-66.889,-176.481,6.915,148.253
C08787=1219.569,296.312,-66.860,-176.484,6.912,148.253
C08788=1219.573,296.063,-66.830,-176.486,6.909,148.253
C08789=1219.577,295.815,-66.801,-176.489,6.907,148.253
C08790=1219.581,295.567,-66.772,-176.491,6.904,148.253
C08791=1219.586,295.319,-66.743,-176.493,6.902,148.253
C08792=1219.591,295.070,-66.714,-176.496,6.899,148.253
C08793=1219.595,294.822,-66.684,-176.498,6.897,148.253
C08794=1219.599,294.574,-66.655,-176.501,6.895,148.254
C08795=1219.603,294.326,-66.627,-176.503,6.892,148.254
C08796=1219.608,294.078,-66.598,-176.505,6.890,148.254
C08797=1219.612,293.829,-66.568,-176.508,6.887,148.254
C08798=1219.616,293.580,-66.539,-176.510,6.885,148.254
C08799=1219.620,293.332,-66.510,-176.513,6.883,148.254
C08800=1219.625,293.085,-66.481,-176.515,6.880,148.254
C08801=1219.630,292.836,-66.452,-176.518,6.877,148.254
C08802=1219.633,292.588,-66.423,-176.520,6.875,148.254
C08803=1219.638,292.339,-66.395,-176.522,6.872,148.254
C08804=1219.642,292.091,-66.365,-176.525,6.870,148.254
C08805=1219.647,291.843,-66.336,-176.527,6.868,148.254
C08806=1219.651,291.594,-66.307,-176.530,6.865,148.254
C08807=1219.655,291.346,-66.278,-176.532,6.863,148.255
C08808=1219.660,291.098,-66.250,-176.534,6.861,148.255
C08809=1219.664,290.850,-66.221,-176.537,6.858,148.255
C08810=1219.668,290.601,-66.192,-176.539,6.856,148.255
C08811=1219.673,290.353,-66.163,-176.541,6.853,148.255
C08812=1219.677,290.105,-66.135,-176.544,6.851,148.255
C08813=1219.681,289.856,-66.105,-176.547,6.849,148.255
C08814=1219.686,289.582,-66.073,-176.549,6.846,148.255
C08815=1219.691,289.308,-66.042,-176.552,6.843,148.256
C08816=1219.695,289.034,-66.010,-176.555,6.841,148.256
C08817=1219.700,288.760,-65.978,-176.557,6.838,148.256
C08818=1219.705,288.511,-65.949,-176.560,6.836,148.256
C08819=1219.709,288.263,-65.920,-176.562,6.833,148.256
C08820=1219.713,288.015,-65.892,-176.565,6.830,148.256
C08821=1219.718,287.767,-65.863,-176.567,6.828,148.256
C08822=1219.722,287.518,-65.834,-176.570,6.825,148.256
C08823=1219.726,287.270,-65.806,-176.572,6.823,148.256
C08824=1219.731,287.022,-65.777,-176.574,6.821,148.256
C08825=1219.735,286.773,-65.748,-176.577,6.818,148.257
C08826=1219.739,286.525,-65.720,-176.579,6.816,148.257
C08827=1219.744,286.277,-65.691,-176.581,6.814,148.257
C08828=1219.748,286.028,-65.662,-176.585,6.811,148.257
C08829=1219.753,285.780,-65.634,-176.587,6.809,148.257
C08830=1219.757,285.532,-65.605,-176.589,6.807,148.257
C08831=1219.762,285.284,-65.577,-176.591,6.805,148.257
C08832=1219.766,285.035,-65.548,-176.594,6.802,148.257
C08833=1219.770,284.786,-65.520,-176.596,6.800,148.258
C08834=1219.774,284.539,-65.491,-176.599,6.798,148.258
C08835=1219.779,284.290,-65.462,-176.602,6.795,148.258
C08836=1219.784,284.042,-65.434,-176.604,6.792,148.258
C08837=1219.787,283.793,-65.406,-176.606,6.791,148.258
C08838=1219.792,283.544,-65.377,-176.609,6.788,148.258
C08839=1219.796,283.297,-65.349,-176.611,6.785,148.258
C08840=1219.800,283.048,-65.320,-176.614,6.783,148.259
C08841=1219.805,282.800,-65.292,-176.616,6.780,148.259
C08842=1219.809,282.552,-65.263,-176.618,6.778,148.259
C08843=1219.814,282.304,-65.236,-176.621,6.776,148.259
C08844=1219.818,282.055,-65.207,-176.624,6.773,148.259
C08845=1219.822,281.807,-65.178,-176.626,6.771,148.259
C08846=1219.827,281.559,-65.150,-176.628,6.769,148.259
C08847=1219.830,281.310,-65.122,-176.631,6.767,148.259
C08848=1219.835,281.062,-65.093,-176.634,6.764,148.260
C08849=1219.839,280.813,-65.065,-176.636,6.762,148.260
C08850=1219.844,280.565,-65.037,-176.638,6.760,148.260
C08851=1219.848,280.317,-65.009,-176.641,6.757,148.260
C08852=1219.853,280.068,-64.980,-176.643,6.755,148.260
C08853=1219.857,279.820,-64.952,-176.645,6.753,148.260
C08854=1219.862,279.572,-64.924,-176.648,6.751,148.260
C08855=1219.866,279.323,-64.895,-176.651,6.748,148.260
C08856=1219.871,279.075,-64.867,-176.653,6.746,148.261
C08857=1219.875,278.826,-64.839,-176.655,6.744,148.261
C08858=1219.879,278.578,-64.811,-176.658,6.741,148.261
C08859=1219.883,278.330,-64.782,-176.661,6.739,148.261
C08860=1219.888,278.082,-64.755,-176.663,6.737,148.261
C08861=1219.892,277.833,-64.727,-176.665,6.735,148.262
C08862=1219.897,277.585,-64.698,-176.668,6.732,148.262
C08863=1219.900,277.336,-64.670,-176.670,6.729,148.262
C08864=1219.905,277.088,-64.642,-176.673,6.728,148.262
C08865=1219.909,276.839,-64.614,-176.675,6.725,148.262
C08866=1219.914,276.591,-64.586,-176.678,6.723,148.262
C08867=1219.918,276.342,-64.558,-176.680,6.720,148.262
C08868=1219.923,276.094,-64.530,-176.683,6.719,148.263
C08869=1219.927,275.846,-64.502,-176.685,6.716,148.263
C08870=1219.932,275.598,-64.473,-176.688,6.713,148.263
C08871=1219.936,275.349,-64.446,-176.690,6.711,148.263
C08872=1219.940,275.100,-64.418,-176.692,6.709,148.263
C08873=1219.945,274.852,-64.390,-176.695,6.707,148.263
C08874=1219.949,274.604,-64.362,-176.698,6.704,148.263
C08875=1219.953,274.356,-64.334,-176.700,6.702,148.264
C08876=1219.958,274.107,-64.307,-176.702,6.700,148.264
C08877=1219.962,273.858,-64.278,-176.705,6.698,148.264
C08878=1219.967,273.611,-64.250,-176.708,6.695,148.264
C08879=1219.970,273.362,-64.222,-176.710,6.693,148.264
C08880=1219.975,273.113,-64.195,-176.712,6.691,148.264
C08881=1219.980,272.865,-64.167,-176.715,6.688,148.265
C08882=1219.984,272.617,-64.139,-176.718,6.686,148.265
C08883=1219.989,272.368,-64.112,-176.720,6.684,148.265
C08884=1219.992,272.120,-64.083,-176.722,6.682,148.265
C08885=1219.997,271.871,-64.055,-176.725,6.679,148.265
C08886=1220.002,271.623,-64.028,-176.728,6.677,148.265
C08887=1220.006,271.374,-64.000,-176.730,6.675,148.266
C08888=1220.010,271.127,-63.972,-176.732,6.673,148.266
C08889=1220.015,270.878,-63.945,-176.734,6.671,148.266
C08890=1220.019,270.629,-63.917,-176.738,6.668,148.266
C08891=1220.024,270.381,-63.889,-176.740,6.666,148.266
C08892=1220.028,270.133,-63.861,-176.742,6.664,148.267
C08893=1220.032,269.884,-63.834,-176.744,6.662,148.267
C08894=1220.037,269.636,-63.806,-176.748,6.659,148.267
C08895=1220.041,269.388,-63.778,-176.750,6.657,148.267
C08896=1220.045,269.139,-63.751,-176.752,6.655,148.267
C08897=1220.049,268.891,-63.723,-176.755,6.653,148.267
C08898=1220.055,268.642,-63.696,-176.758,6.650,148.268
C08899=1220.059,268.393,-63.667,-176.760,6.648,148.268
C08900=1220.063,268.145,-63.640,-176.762,6.646,148.268
C08901=1220.068,267.897,-63.613,-176.765,6.644,148.268
C08902=1220.072,267.649,-63.586,-176.767,6.642,148.268
C08903=1220.076,267.399,-63.558,-176.770,6.639,148.269
C08904=1220.081,267.151,-63.530,-176.772,6.637,148.269
C08905=1220.085,266.903,-63.503,-176.775,6.635,148.269
C08906=1220.089,266.654,-63.475,-176.777,6.633,148.269
C08907=1220.094,266.406,-63.448,-176.780,6.631,148.269
C08908=1220.098,266.157,-63.421,-176.782,6.628,148.269
C08909=1220.103,265.909,-63.393,-176.785,6.626,148.270
C08910=1220.107,265.660,-63.366,-176.787,6.624,148.270
C08911=1220.111,265.412,-63.338,-176.790,6.622,148.270
C08912=1220.116,265.164,-63.311,-176.792,6.620,148.270
C08913=1220.120,264.915,-63.284,-176.795,6.617,148.270
C08914=1220.124,264.667,-63.256,-176.797,6.615,148.270
C08915=1220.129,264.418,-63.229,-176.800,6.613,148.271
C08916=1220.133,264.170,-63.202,-176.802,6.611,148.271
C08917=1220.138,263.921,-63.175,-176.805,6.609,148.271
C08918=1220.143,263.649,-63.144,-176.808,6.606,148.271
C08919=1220.147,263.376,-63.114,-176.810,6.605,148.272
C08920=1220.153,263.103,-63.084,-176.813,6.602,148.272
C08921=1220.157,262.831,-63.054,-176.816,6.600,148.272
C08922=1220.162,262.582,-63.027,-176.819,6.597,148.272
C08923=1220.166,262.334,-63.000,-176.821,6.595,148.272
C08924=1220.171,262.085,-62.973,-176.823,6.593,148.273
C08925=1220.175,261.837,-62.945,-176.826,6.591,148.273
C08926=1220.179,261.588,-62.918,-176.828,6.589,148.273
C08927=1220.184,261.340,-62.891,-176.831,6.587,148.273
C08928=1220.188,261.092,-62.864,-176.834,6.584,148.273
C08929=1220.193,260.843,-62.837,-176.836,6.582,148.274
C08930=1220.197,260.595,-62.810,-176.838,6.580,148.274
C08931=1220.201,260.346,-62.782,-176.841,6.578,148.274
C08932=1220.206,260.097,-62.755,-176.843,6.576,148.274
C08933=1220.210,259.849,-62.728,-176.846,6.574,148.274
C08934=1220.215,259.601,-62.701,-176.849,6.571,148.275
C08935=1220.219,259.352,-62.674,-176.851,6.569,148.275
C08936=1220.224,259.104,-62.647,-176.854,6.567,148.275
C08937=1220.228,258.855,-62.620,-176.856,6.565,148.275
C08938=1220.232,258.606,-62.593,-176.858,6.563,148.275
C08939=1220.237,258.358,-62.566,-176.861,6.561,148.276
C08940=1220.241,258.109,-62.539,-176.863,6.559,148.276
C08941=1220.246,257.861,-62.512,-176.866,6.556,148.276
C08942=1220.250,257.612,-62.485,-176.869,6.554,148.276
C08943=1220.255,257.364,-62.458,-176.871,6.552,148.277
C08944=1220.260,257.115,-62.431,-176.874,6.550,148.277
C08945=1220.264,256.867,-62.405,-176.876,6.548,148.277
C08946=1220.268,256.619,-62.377,-176.878,6.546,148.277
C08947=1220.272,256.370,-62.350,-176.881,6.543,148.277
C08948=1220.277,256.121,-62.323,-176.884,6.541,148.278
C08949=1220.281,255.873,-62.297,-176.886,6.539,148.278
C08950=1220.285,255.624,-62.269,-176.889,6.538,148.278
C08951=1220.290,255.376,-62.242,-176.891,6.535,148.278
C08952=1220.294,255.127,-62.217,-176.894,6.533,148.279
C08953=1220.299,254.879,-62.190,-176.896,6.532,148.279
C08954=1220.304,254.630,-62.163,-176.898,6.529,148.279
C08955=1220.308,254.382,-62.136,-176.901,6.527,148.279
C08956=1220.312,254.133,-62.109,-176.904,6.525,148.280
C08957=1220.317,253.885,-62.082,-176.906,6.523,148.280
C08958=1220.321,253.637,-62.055,-176.909,6.521,148.280
C08959=1220.326,253.388,-62.029,-176.911,6.519,148.280
C08960=1220.330,253.139,-62.002,-176.914,6.517,148.280
C08961=1220.334,252.891,-61.976,-176.916,6.515,148.281
C08962=1220.339,252.642,-61.949,-176.919,6.513,148.281
C08963=1220.344,252.393,-61.922,-176.921,6.510,148.281
C08964=1220.348,252.145,-61.896,-176.924,6.508,148.281
C08965=1220.353,251.897,-61.869,-176.927,6.506,148.282
C08966=1220.356,251.648,-61.842,-176.929,6.504,148.282
C08967=1220.361,251.399,-61.816,-176.931,6.502,148.282
C08968=1220.366,251.151,-61.789,-176.934,6.500,148.282
C08969=1220.370,250.903,-61.762,-176.936,6.498,148.282
C08970=1220.375,250.654,-61.736,-176.939,6.496,148.283
C08971=1220.379,250.405,-61.709,-176.941,6.494,148.283
C08972=1220.384,250.157,-61.682,-176.944,6.492,148.283
C08973=1220.388,249.908,-61.657,-176.947,6.489,148.283
C08974=1220.392,249.660,-61.630,-176.949,6.487,148.284
C08975=1220.396,249.411,-61.603,-176.951,6.485,148.284
C08976=1220.401,249.162,-61.577,-176.954,6.483,148.284
C08977=1220.406,248.914,-61.550,-176.957,6.482,148.284
C08978=1220.410,248.666,-61.523,-176.959,6.480,148.285
C08979=1220.415,248.416,-61.497,-176.961,6.477,148.285
C08980=1220.419,248.168,-61.470,-176.964,6.476,148.285
C08981=1220.423,247.920,-61.445,-176.967,6.474,148.285
C08982=1220.428,247.671,-61.418,-176.969,6.472,148.285
C08983=1220.432,247.422,-61.392,-176.972,6.469,148.286
C08984=1220.437,247.174,-61.365,-176.975,6.467,148.286
C08985=1220.441,246.926,-61.339,-176.977,6.465,148.286
C08986=1220.446,246.677,-61.312,-176.979,6.463,148.286
C08987=1220.450,246.428,-61.287,-176.982,6.461,148.287
C08988=1220.455,246.180,-61.260,-176.985,6.459,148.287
C08989=1220.459,245.931,-61.234,-176.987,6.457,148.287
C08990=1220.464,245.683,-61.207,-176.989,6.455,148.287
C08991=1220.468,245.434,-61.181,-176.992,6.453,148.288
C08992=1220.472,245.186,-61.155,-176.995,6.451,148.288
C08993=1220.477,244.936,-61.128,-176.997,6.449,148.288
C08994=1220.482,244.688,-61.103,-176.999,6.447,148.289
C08995=1220.486,244.440,-61.076,-177.002,6.445,148.289
C08996=1220.491,244.191,-61.050,-177.005,6.444,148.289
C08997=1220.494,243.943,-61.024,-177.007,6.441,148.289
C08998=1220.499,243.694,-60.997,-177.010,6.439,148.290
C08999=1220.504,243.445,-60.971,-177.012,6.437,148.290
C09000=1220.508,243.197,-60.945,-177.015,6.435,148.290
C09001=1220.513,242.948,-60.919,-177.017,6.433,148.290
C09002=1220.517,242.700,-60.893,-177.020,6.431,148.291
C09003=1220.521,242.451,-60.867,-177.022,6.429,148.291
C09004=1220.526,242.202,-60.840,-177.025,6.427,148.291
C09005=1220.530,241.953,-60.815,-177.027,6.425,148.291
C09006=1220.534,241.705,-60.788,-177.030,6.423,148.292
C09007=1220.540,241.457,-60.762,-177.032,6.421,148.292
C09008=1220.544,241.208,-60.736,-177.035,6.419,148.292
C09009=1220.548,240.959,-60.711,-177.037,6.417,148.292
C09010=1220.552,240.711,-60.684,-177.040,6.415,148.293
C09011=1220.557,240.462,-60.658,-177.042,6.413,148.293
C09012=1220.562,240.214,-60.633,-177.045,6.412,148.293
C09013=1220.566,239.965,-60.607,-177.047,6.409,148.293
C09014=1220.571,239.716,-60.581,-177.050,6.408,148.294
C09015=1220.575,239.468,-60.554,-177.052,6.406,148.294
C09016=1220.580,239.220,-60.529,-177.055,6.404,148.294
C09017=1220.584,238.971,-60.503,-177.058,6.402,148.295
C09018=1220.589,238.722,-60.477,-177.060,6.400,148.295
C09019=1220.593,238.473,-60.451,-177.063,6.397,148.295
C09020=1220.598,238.224,-60.425,-177.066,6.395,148.295
C09021=1220.603,237.976,-60.400,-177.068,6.393,148.296
C09022=1220.607,237.705,-60.371,-177.071,6.391,148.296
C09023=1220.612,237.433,-60.343,-177.074,6.390,148.296
C09024=1220.617,237.162,-60.315,-177.076,6.388,148.297
C09025=1220.621,236.890,-60.286,-177.079,6.385,148.297
C09026=1220.626,236.642,-60.261,-177.081,6.383,148.297
C09027=1220.631,236.393,-60.235,-177.084,6.381,148.297
C09028=1220.635,236.144,-60.209,-177.087,6.379,148.298
C09029=1220.640,235.895,-60.183,-177.089,6.377,148.298
C09030=1220.644,235.647,-60.158,-177.092,6.375,148.298
C09031=1220.649,235.399,-60.132,-177.094,6.373,148.298
C09032=1220.653,235.150,-60.106,-177.097,6.371,148.299
C09033=1220.658,234.902,-60.081,-177.099,6.369,148.299
C09034=1220.662,234.653,-60.055,-177.102,6.368,148.299
C09035=1220.666,234.404,-60.029,-177.105,6.366,148.300
C09036=1220.672,234.156,-60.003,-177.107,6.363,148.300
C09037=1220.676,233.907,-59.978,-177.109,6.362,148.300
C09038=1220.680,233.658,-59.952,-177.112,6.360,148.300
C09039=1220.685,233.410,-59.927,-177.115,6.358,148.301
C09040=1220.689,233.160,-59.901,-177.117,6.356,148.301
C09041=1220.694,232.912,-59.876,-177.120,6.354,148.301
C09042=1220.698,232.664,-59.850,-177.122,6.352,148.301
C09043=1220.703,232.415,-59.825,-177.125,6.350,148.302
C09044=1220.707,232.166,-59.799,-177.127,6.348,148.302
C09045=1220.712,231.918,-59.773,-177.130,6.346,148.302
C09046=1220.716,231.669,-59.748,-177.132,6.345,148.303
C09047=1220.721,231.420,-59.723,-177.135,6.343,148.303
C09048=1220.725,231.172,-59.697,-177.137,6.340,148.303
C09049=1220.730,230.923,-59.672,-177.140,6.339,148.303
C09050=1220.734,230.675,-59.646,-177.142,6.337,148.304
C09051=1220.739,230.426,-59.620,-177.145,6.335,148.304
C09052=1220.743,230.176,-59.595,-177.148,6.333,148.304
C09053=1220.748,229.928,-59.570,-177.150,6.331,148.305
C09054=1220.752,229.679,-59.544,-177.153,6.329,148.305
C09055=1220.756,229.431,-59.518,-177.155,6.327,148.305
C09056=1220.762,229.182,-59.494,-177.158,6.325,148.305
C09057=1220.766,228.933,-59.468,-177.160,6.323,148.306
C09058=1220.770,228.685,-59.443,-177.163,6.322,148.306
C09059=1220.774,228.436,-59.418,-177.166,6.320,148.306
C09060=1220.779,228.188,-59.393,-177.168,6.318,148.307
C09061=1220.783,227.939,-59.367,-177.171,6.316,148.307
C09062=1220.788,227.690,-59.342,-177.174,6.314,148.307
C09063=1220.793,227.441,-59.317,-177.176,6.312,148.307
C09064=1220.797,227.193,-59.291,-177.178,6.310,148.308
C09065=1220.802,226.944,-59.266,-177.181,6.308,148.308
C09066=1220.806,226.695,-59.241,-177.184,6.306,148.308
C09067=1220.810,226.447,-59.216,-177.186,6.304,148.309
C09068=1220.815,226.198,-59.191,-177.189,6.303,148.309
C09069=1220.820,225.950,-59.165,-177.191,6.302,148.309
C09070=1220.824,225.700,-59.140,-177.194,6.300,148.310
C09071=1220.829,225.452,-59.115,-177.196,6.298,148.310
C09072=1220.834,225.203,-59.090,-177.198,6.296,148.310
C09073=1220.837,224.954,-59.065,-177.201,6.294,148.311
C09074=1220.842,224.706,-59.039,-177.204,6.292,148.311
C09075=1220.847,224.457,-59.014,-177.206,6.290,148.311
C09076=1220.851,224.209,-58.989,-177.209,6.288,148.312
C09077=1220.856,223.959,-58.964,-177.211,6.286,148.312
C09078=1220.860,223.712,-58.939,-177.214,6.285,148.312
C09079=1220.865,223.462,-58.914,-177.217,6.283,148.312
C09080=1220.870,223.213,-58.889,-177.219,6.281,148.313
C09081=1220.875,222.965,-58.864,-177.221,6.279,148.313
C09082=1220.878,222.716,-58.840,-177.224,6.277,148.313
C09083=1220.883,222.468,-58.814,-177.227,6.275,148.314
C09084=1220.888,222.219,-58.789,-177.229,6.273,148.314
C09085=1220.892,221.971,-58.764,-177.232,6.271,148.314
C09086=1220.896,221.721,-58.739,-177.235,6.269,148.315
C09087=1220.901,221.473,-58.715,-177.237,6.268,148.315
C09088=1220.906,221.224,-58.689,-177.240,6.266,148.315
C09089=1220.910,220.975,-58.665,-177.242,6.264,148.316
C09090=1220.915,220.726,-58.640,-177.245,6.262,148.316
C09091=1220.919,220.478,-58.614,-177.247,6.261,148.316
C09092=1220.923,220.229,-58.590,-177.250,6.259,148.317
C09093=1220.928,219.980,-58.565,-177.252,6.257,148.317
C09094=1220.933,219.732,-58.540,-177.255,6.255,148.317
C09095=1220.937,219.483,-58.515,-177.257,6.253,148.317
C09096=1220.942,219.234,-58.491,-177.260,6.251,148.318
C09097=1220.946,218.985,-58.465,-177.262,6.249,148.318
C09098=1220.951,218.737,-58.441,-177.265,6.248,148.318
C09099=1220.956,218.488,-58.416,-177.268,6.246,148.319
C09100=1220.960,218.239,-58.392,-177.270,6.244,148.319
C09101=1220.964,217.991,-58.366,-177.273,6.242,148.319
C09102=1220.969,217.742,-58.341,-177.276,6.240,148.320
C09103=1220.973,217.493,-58.317,-177.278,6.238,148.320
C09104=1220.978,217.244,-58.293,-177.281,6.236,148.320
C09105=1220.982,216.995,-58.268,-177.284,6.235,148.321
C09106=1220.987,216.747,-58.243,-177.286,6.233,148.321
C09107=1220.992,216.499,-58.218,-177.288,6.232,148.321
C09108=1220.996,216.249,-58.194,-177.291,6.230,148.322
C09109=1221.001,216.001,-58.169,-177.294,6.228,148.322
C09110=1221.005,215.752,-58.145,-177.296,6.226,148.322
C09111=1221.010,215.503,-58.120,-177.299,6.224,148.323
C09112=1221.014,215.254,-58.096,-177.301,6.222,148.323
C09113=1221.019,215.006,-58.070,-177.304,6.221,148.323
C09114=1221.023,214.757,-58.046,-177.307,6.219,148.324
C09115=1221.028,214.509,-58.021,-177.309,6.217,148.324
C09116=1221.032,214.259,-57.997,-177.312,6.215,148.324
C09117=1221.037,214.011,-57.972,-177.315,6.213,148.325
C09118=1221.042,213.762,-57.948,-177.317,6.211,148.325
C09119=1221.046,213.513,-57.923,-177.319,6.210,148.325
C09120=1221.050,213.264,-57.899,-177.322,6.208,148.326
C09121=1221.056,213.016,-57.874,-177.325,6.207,148.326
C09122=1221.060,212.767,-57.850,-177.327,6.205,148.326
C09123=1221.065,212.518,-57.825,-177.330,6.203,148.327
C09124=1221.069,212.269,-57.801,-177.332,6.201,148.327
C09125=1221.073,212.021,-57.777,-177.335,6.199,148.327
C09126=1221.078,211.750,-57.750,-177.338,6.197,148.328
C09127=1221.083,211.479,-57.724,-177.340,6.196,148.328
C09128=1221.088,211.209,-57.697,-177.343,6.194,148.328
C09129=1221.094,210.939,-57.671,-177.346,6.191,148.329
